   // UNICODE_TO_GBK[4694] := 16#545E;
   // UNICODE_TO_GBK[4695] := 16#85DA;
   // UNICODE_TO_GBK[4696] := 16#545F;
   // UNICODE_TO_GBK[4697] := 16#85DB;
   // UNICODE_TO_GBK[4698] := 16#5460;
   // UNICODE_TO_GBK[4699] := 16#85DC;
   // UNICODE_TO_GBK[4700] := 16#5461;
   // UNICODE_TO_GBK[4701] := 16#85DD;
   // UNICODE_TO_GBK[4702] := 16#5462;
   // UNICODE_TO_GBK[4703] := 16#C4D8;
   // UNICODE_TO_GBK[4704] := 16#5463;
   // UNICODE_TO_GBK[4705] := 16#85DE;
   // UNICODE_TO_GBK[4706] := 16#5464;
   // UNICODE_TO_GBK[4707] := 16#DFCA;
   // UNICODE_TO_GBK[4708] := 16#5465;
   // UNICODE_TO_GBK[4709] := 16#85DF;
   // UNICODE_TO_GBK[4710] := 16#5466;
   // UNICODE_TO_GBK[4711] := 16#DFCF;
   // UNICODE_TO_GBK[4712] := 16#5467;
   // UNICODE_TO_GBK[4713] := 16#85E0;
   // UNICODE_TO_GBK[4714] := 16#5468;
   // UNICODE_TO_GBK[4715] := 16#D6DC;
   // UNICODE_TO_GBK[4716] := 16#5469;
   // UNICODE_TO_GBK[4717] := 16#85E1;
   // UNICODE_TO_GBK[4718] := 16#546A;
   // UNICODE_TO_GBK[4719] := 16#85E2;
   // UNICODE_TO_GBK[4720] := 16#546B;
   // UNICODE_TO_GBK[4721] := 16#85E3;
   // UNICODE_TO_GBK[4722] := 16#546C;
   // UNICODE_TO_GBK[4723] := 16#85E4;
   // UNICODE_TO_GBK[4724] := 16#546D;
   // UNICODE_TO_GBK[4725] := 16#85E5;
   // UNICODE_TO_GBK[4726] := 16#546E;
   // UNICODE_TO_GBK[4727] := 16#85E6;
   // UNICODE_TO_GBK[4728] := 16#546F;
   // UNICODE_TO_GBK[4729] := 16#85E7;
   // UNICODE_TO_GBK[4730] := 16#5470;
   // UNICODE_TO_GBK[4731] := 16#85E8;
   // UNICODE_TO_GBK[4732] := 16#5471;
   // UNICODE_TO_GBK[4733] := 16#DFC9;
   // UNICODE_TO_GBK[4734] := 16#5472;
   // UNICODE_TO_GBK[4735] := 16#DFDA;
   // UNICODE_TO_GBK[4736] := 16#5473;
   // UNICODE_TO_GBK[4737] := 16#CEB6;
   // UNICODE_TO_GBK[4738] := 16#5474;
   // UNICODE_TO_GBK[4739] := 16#85E9;
   // UNICODE_TO_GBK[4740] := 16#5475;
   // UNICODE_TO_GBK[4741] := 16#BAC7;
   // UNICODE_TO_GBK[4742] := 16#5476;
   // UNICODE_TO_GBK[4743] := 16#DFCE;
   // UNICODE_TO_GBK[4744] := 16#5477;
   // UNICODE_TO_GBK[4745] := 16#DFC8;
   // UNICODE_TO_GBK[4746] := 16#5478;
   // UNICODE_TO_GBK[4747] := 16#C5DE;
   // UNICODE_TO_GBK[4748] := 16#5479;
   // UNICODE_TO_GBK[4749] := 16#85EA;
   // UNICODE_TO_GBK[4750] := 16#547A;
   // UNICODE_TO_GBK[4751] := 16#85EB;
   // UNICODE_TO_GBK[4752] := 16#547B;
   // UNICODE_TO_GBK[4753] := 16#C9EB;
   // UNICODE_TO_GBK[4754] := 16#547C;
   // UNICODE_TO_GBK[4755] := 16#BAF4;
   // UNICODE_TO_GBK[4756] := 16#547D;
   // UNICODE_TO_GBK[4757] := 16#C3FC;
   // UNICODE_TO_GBK[4758] := 16#547E;
   // UNICODE_TO_GBK[4759] := 16#85EC;
   // UNICODE_TO_GBK[4760] := 16#547F;
   // UNICODE_TO_GBK[4761] := 16#85ED;
   // UNICODE_TO_GBK[4762] := 16#5480;
   // UNICODE_TO_GBK[4763] := 16#BED7;
   // UNICODE_TO_GBK[4764] := 16#5481;
   // UNICODE_TO_GBK[4765] := 16#85EE;
   // UNICODE_TO_GBK[4766] := 16#5482;
   // UNICODE_TO_GBK[4767] := 16#DFC6;
   // UNICODE_TO_GBK[4768] := 16#5483;
   // UNICODE_TO_GBK[4769] := 16#85EF;
   // UNICODE_TO_GBK[4770] := 16#5484;
   // UNICODE_TO_GBK[4771] := 16#DFCD;
   // UNICODE_TO_GBK[4772] := 16#5485;
   // UNICODE_TO_GBK[4773] := 16#85F0;
   // UNICODE_TO_GBK[4774] := 16#5486;
   // UNICODE_TO_GBK[4775] := 16#C5D8;
   // UNICODE_TO_GBK[4776] := 16#5487;
   // UNICODE_TO_GBK[4777] := 16#85F1;
   // UNICODE_TO_GBK[4778] := 16#5488;
   // UNICODE_TO_GBK[4779] := 16#85F2;
   // UNICODE_TO_GBK[4780] := 16#5489;
   // UNICODE_TO_GBK[4781] := 16#85F3;
   // UNICODE_TO_GBK[4782] := 16#548A;
   // UNICODE_TO_GBK[4783] := 16#85F4;
   // UNICODE_TO_GBK[4784] := 16#548B;
   // UNICODE_TO_GBK[4785] := 16#D5A6;
   // UNICODE_TO_GBK[4786] := 16#548C;
   // UNICODE_TO_GBK[4787] := 16#BACD;
   // UNICODE_TO_GBK[4788] := 16#548D;
   // UNICODE_TO_GBK[4789] := 16#85F5;
   // UNICODE_TO_GBK[4790] := 16#548E;
   // UNICODE_TO_GBK[4791] := 16#BECC;
   // UNICODE_TO_GBK[4792] := 16#548F;
   // UNICODE_TO_GBK[4793] := 16#D3BD;
   // UNICODE_TO_GBK[4794] := 16#5490;
   // UNICODE_TO_GBK[4795] := 16#B8C0;
   // UNICODE_TO_GBK[4796] := 16#5491;
   // UNICODE_TO_GBK[4797] := 16#85F6;
   // UNICODE_TO_GBK[4798] := 16#5492;
   // UNICODE_TO_GBK[4799] := 16#D6E4;
   // UNICODE_TO_GBK[4800] := 16#5493;
   // UNICODE_TO_GBK[4801] := 16#85F7;
   // UNICODE_TO_GBK[4802] := 16#5494;
   // UNICODE_TO_GBK[4803] := 16#DFC7;
   // UNICODE_TO_GBK[4804] := 16#5495;
   // UNICODE_TO_GBK[4805] := 16#B9BE;
   // UNICODE_TO_GBK[4806] := 16#5496;
   // UNICODE_TO_GBK[4807] := 16#BFA7;
   // UNICODE_TO_GBK[4808] := 16#5497;
   // UNICODE_TO_GBK[4809] := 16#85F8;
   // UNICODE_TO_GBK[4810] := 16#5498;
   // UNICODE_TO_GBK[4811] := 16#85F9;
   // UNICODE_TO_GBK[4812] := 16#5499;
   // UNICODE_TO_GBK[4813] := 16#C1FC;
   // UNICODE_TO_GBK[4814] := 16#549A;
   // UNICODE_TO_GBK[4815] := 16#DFCB;
   // UNICODE_TO_GBK[4816] := 16#549B;
   // UNICODE_TO_GBK[4817] := 16#DFCC;
   // UNICODE_TO_GBK[4818] := 16#549C;
   // UNICODE_TO_GBK[4819] := 16#85FA;
   // UNICODE_TO_GBK[4820] := 16#549D;
   // UNICODE_TO_GBK[4821] := 16#DFD0;
   // UNICODE_TO_GBK[4822] := 16#549E;
   // UNICODE_TO_GBK[4823] := 16#85FB;
   // UNICODE_TO_GBK[4824] := 16#549F;
   // UNICODE_TO_GBK[4825] := 16#85FC;
   // UNICODE_TO_GBK[4826] := 16#54A0;
   // UNICODE_TO_GBK[4827] := 16#85FD;
   // UNICODE_TO_GBK[4828] := 16#54A1;
   // UNICODE_TO_GBK[4829] := 16#85FE;
   // UNICODE_TO_GBK[4830] := 16#54A2;
   // UNICODE_TO_GBK[4831] := 16#8640;
   // UNICODE_TO_GBK[4832] := 16#54A3;
   // UNICODE_TO_GBK[4833] := 16#DFDB;
   // UNICODE_TO_GBK[4834] := 16#54A4;
   // UNICODE_TO_GBK[4835] := 16#DFE5;
   // UNICODE_TO_GBK[4836] := 16#54A5;
   // UNICODE_TO_GBK[4837] := 16#8641;
   // UNICODE_TO_GBK[4838] := 16#54A6;
   // UNICODE_TO_GBK[4839] := 16#DFD7;
   // UNICODE_TO_GBK[4840] := 16#54A7;
   // UNICODE_TO_GBK[4841] := 16#DFD6;
   // UNICODE_TO_GBK[4842] := 16#54A8;
   // UNICODE_TO_GBK[4843] := 16#D7C9;
   // UNICODE_TO_GBK[4844] := 16#54A9;
   // UNICODE_TO_GBK[4845] := 16#DFE3;
   // UNICODE_TO_GBK[4846] := 16#54AA;
   // UNICODE_TO_GBK[4847] := 16#DFE4;
   // UNICODE_TO_GBK[4848] := 16#54AB;
   // UNICODE_TO_GBK[4849] := 16#E5EB;
   // UNICODE_TO_GBK[4850] := 16#54AC;
   // UNICODE_TO_GBK[4851] := 16#D2A7;
   // UNICODE_TO_GBK[4852] := 16#54AD;
   // UNICODE_TO_GBK[4853] := 16#DFD2;
   // UNICODE_TO_GBK[4854] := 16#54AE;
   // UNICODE_TO_GBK[4855] := 16#8642;
   // UNICODE_TO_GBK[4856] := 16#54AF;
   // UNICODE_TO_GBK[4857] := 16#BFA9;
   // UNICODE_TO_GBK[4858] := 16#54B0;
   // UNICODE_TO_GBK[4859] := 16#8643;
   // UNICODE_TO_GBK[4860] := 16#54B1;
   // UNICODE_TO_GBK[4861] := 16#D4DB;
   // UNICODE_TO_GBK[4862] := 16#54B2;
   // UNICODE_TO_GBK[4863] := 16#8644;
   // UNICODE_TO_GBK[4864] := 16#54B3;
   // UNICODE_TO_GBK[4865] := 16#BFC8;
   // UNICODE_TO_GBK[4866] := 16#54B4;
   // UNICODE_TO_GBK[4867] := 16#DFD4;
   // UNICODE_TO_GBK[4868] := 16#54B5;
   // UNICODE_TO_GBK[4869] := 16#8645;
   // UNICODE_TO_GBK[4870] := 16#54B6;
   // UNICODE_TO_GBK[4871] := 16#8646;
   // UNICODE_TO_GBK[4872] := 16#54B7;
   // UNICODE_TO_GBK[4873] := 16#8647;
   // UNICODE_TO_GBK[4874] := 16#54B8;
   // UNICODE_TO_GBK[4875] := 16#CFCC;
   // UNICODE_TO_GBK[4876] := 16#54B9;
   // UNICODE_TO_GBK[4877] := 16#8648;
   // UNICODE_TO_GBK[4878] := 16#54BA;
   // UNICODE_TO_GBK[4879] := 16#8649;
   // UNICODE_TO_GBK[4880] := 16#54BB;
   // UNICODE_TO_GBK[4881] := 16#DFDD;
   // UNICODE_TO_GBK[4882] := 16#54BC;
   // UNICODE_TO_GBK[4883] := 16#864A;
   // UNICODE_TO_GBK[4884] := 16#54BD;
   // UNICODE_TO_GBK[4885] := 16#D1CA;
   // UNICODE_TO_GBK[4886] := 16#54BE;
   // UNICODE_TO_GBK[4887] := 16#864B;
   // UNICODE_TO_GBK[4888] := 16#54BF;
   // UNICODE_TO_GBK[4889] := 16#DFDE;
   // UNICODE_TO_GBK[4890] := 16#54C0;
   // UNICODE_TO_GBK[4891] := 16#B0A7;
   // UNICODE_TO_GBK[4892] := 16#54C1;
   // UNICODE_TO_GBK[4893] := 16#C6B7;
   // UNICODE_TO_GBK[4894] := 16#54C2;
   // UNICODE_TO_GBK[4895] := 16#DFD3;
   // UNICODE_TO_GBK[4896] := 16#54C3;
   // UNICODE_TO_GBK[4897] := 16#864C;
   // UNICODE_TO_GBK[4898] := 16#54C4;
   // UNICODE_TO_GBK[4899] := 16#BAE5;
   // UNICODE_TO_GBK[4900] := 16#54C5;
   // UNICODE_TO_GBK[4901] := 16#864D;
   // UNICODE_TO_GBK[4902] := 16#54C6;
   // UNICODE_TO_GBK[4903] := 16#B6DF;
   // UNICODE_TO_GBK[4904] := 16#54C7;
   // UNICODE_TO_GBK[4905] := 16#CDDB;
   // UNICODE_TO_GBK[4906] := 16#54C8;
   // UNICODE_TO_GBK[4907] := 16#B9FE;
   // UNICODE_TO_GBK[4908] := 16#54C9;
   // UNICODE_TO_GBK[4909] := 16#D4D5;
   // UNICODE_TO_GBK[4910] := 16#54CA;
   // UNICODE_TO_GBK[4911] := 16#864E;
   // UNICODE_TO_GBK[4912] := 16#54CB;
   // UNICODE_TO_GBK[4913] := 16#864F;
   // UNICODE_TO_GBK[4914] := 16#54CC;
   // UNICODE_TO_GBK[4915] := 16#DFDF;
   // UNICODE_TO_GBK[4916] := 16#54CD;
   // UNICODE_TO_GBK[4917] := 16#CFEC;
   // UNICODE_TO_GBK[4918] := 16#54CE;
   // UNICODE_TO_GBK[4919] := 16#B0A5;
   // UNICODE_TO_GBK[4920] := 16#54CF;
   // UNICODE_TO_GBK[4921] := 16#DFE7;
   // UNICODE_TO_GBK[4922] := 16#54D0;
   // UNICODE_TO_GBK[4923] := 16#DFD1;
   // UNICODE_TO_GBK[4924] := 16#54D1;
   // UNICODE_TO_GBK[4925] := 16#D1C6;
   // UNICODE_TO_GBK[4926] := 16#54D2;
   // UNICODE_TO_GBK[4927] := 16#DFD5;
   // UNICODE_TO_GBK[4928] := 16#54D3;
   // UNICODE_TO_GBK[4929] := 16#DFD8;
   // UNICODE_TO_GBK[4930] := 16#54D4;
   // UNICODE_TO_GBK[4931] := 16#DFD9;
   // UNICODE_TO_GBK[4932] := 16#54D5;
   // UNICODE_TO_GBK[4933] := 16#DFDC;
   // UNICODE_TO_GBK[4934] := 16#54D6;
   // UNICODE_TO_GBK[4935] := 16#8650;
   // UNICODE_TO_GBK[4936] := 16#54D7;
   // UNICODE_TO_GBK[4937] := 16#BBA9;
   // UNICODE_TO_GBK[4938] := 16#54D8;
   // UNICODE_TO_GBK[4939] := 16#8651;
   // UNICODE_TO_GBK[4940] := 16#54D9;
   // UNICODE_TO_GBK[4941] := 16#DFE0;
   // UNICODE_TO_GBK[4942] := 16#54DA;
   // UNICODE_TO_GBK[4943] := 16#DFE1;
   // UNICODE_TO_GBK[4944] := 16#54DB;
   // UNICODE_TO_GBK[4945] := 16#8652;
   // UNICODE_TO_GBK[4946] := 16#54DC;
   // UNICODE_TO_GBK[4947] := 16#DFE2;
   // UNICODE_TO_GBK[4948] := 16#54DD;
   // UNICODE_TO_GBK[4949] := 16#DFE6;
   // UNICODE_TO_GBK[4950] := 16#54DE;
   // UNICODE_TO_GBK[4951] := 16#DFE8;
   // UNICODE_TO_GBK[4952] := 16#54DF;
   // UNICODE_TO_GBK[4953] := 16#D3B4;
   // UNICODE_TO_GBK[4954] := 16#54E0;
   // UNICODE_TO_GBK[4955] := 16#8653;
   // UNICODE_TO_GBK[4956] := 16#54E1;
   // UNICODE_TO_GBK[4957] := 16#8654;
   // UNICODE_TO_GBK[4958] := 16#54E2;
   // UNICODE_TO_GBK[4959] := 16#8655;
   // UNICODE_TO_GBK[4960] := 16#54E3;
   // UNICODE_TO_GBK[4961] := 16#8656;
   // UNICODE_TO_GBK[4962] := 16#54E4;
   // UNICODE_TO_GBK[4963] := 16#8657;
   // UNICODE_TO_GBK[4964] := 16#54E5;
   // UNICODE_TO_GBK[4965] := 16#B8E7;
   // UNICODE_TO_GBK[4966] := 16#54E6;
   // UNICODE_TO_GBK[4967] := 16#C5B6;
   // UNICODE_TO_GBK[4968] := 16#54E7;
   // UNICODE_TO_GBK[4969] := 16#DFEA;
   // UNICODE_TO_GBK[4970] := 16#54E8;
   // UNICODE_TO_GBK[4971] := 16#C9DA;
   // UNICODE_TO_GBK[4972] := 16#54E9;
   // UNICODE_TO_GBK[4973] := 16#C1A8;
   // UNICODE_TO_GBK[4974] := 16#54EA;
   // UNICODE_TO_GBK[4975] := 16#C4C4;
   // UNICODE_TO_GBK[4976] := 16#54EB;
   // UNICODE_TO_GBK[4977] := 16#8658;
   // UNICODE_TO_GBK[4978] := 16#54EC;
   // UNICODE_TO_GBK[4979] := 16#8659;
   // UNICODE_TO_GBK[4980] := 16#54ED;
   // UNICODE_TO_GBK[4981] := 16#BFDE;
   // UNICODE_TO_GBK[4982] := 16#54EE;
   // UNICODE_TO_GBK[4983] := 16#CFF8;
   // UNICODE_TO_GBK[4984] := 16#54EF;
   // UNICODE_TO_GBK[4985] := 16#865A;
   // UNICODE_TO_GBK[4986] := 16#54F0;
   // UNICODE_TO_GBK[4987] := 16#865B;
   // UNICODE_TO_GBK[4988] := 16#54F1;
   // UNICODE_TO_GBK[4989] := 16#865C;
   // UNICODE_TO_GBK[4990] := 16#54F2;
   // UNICODE_TO_GBK[4991] := 16#D5DC;
   // UNICODE_TO_GBK[4992] := 16#54F3;
   // UNICODE_TO_GBK[4993] := 16#DFEE;
   // UNICODE_TO_GBK[4994] := 16#54F4;
   // UNICODE_TO_GBK[4995] := 16#865D;
   // UNICODE_TO_GBK[4996] := 16#54F5;
   // UNICODE_TO_GBK[4997] := 16#865E;
   // UNICODE_TO_GBK[4998] := 16#54F6;
   // UNICODE_TO_GBK[4999] := 16#865F;
   // UNICODE_TO_GBK[5000] := 16#54F7;
   // UNICODE_TO_GBK[5001] := 16#8660;
   // UNICODE_TO_GBK[5002] := 16#54F8;
   // UNICODE_TO_GBK[5003] := 16#8661;
   // UNICODE_TO_GBK[5004] := 16#54F9;
   // UNICODE_TO_GBK[5005] := 16#8662;
   // UNICODE_TO_GBK[5006] := 16#54FA;
   // UNICODE_TO_GBK[5007] := 16#B2B8;
   // UNICODE_TO_GBK[5008] := 16#54FB;
   // UNICODE_TO_GBK[5009] := 16#8663;
   // UNICODE_TO_GBK[5010] := 16#54FC;
   // UNICODE_TO_GBK[5011] := 16#BADF;
   // UNICODE_TO_GBK[5012] := 16#54FD;
   // UNICODE_TO_GBK[5013] := 16#DFEC;
   // UNICODE_TO_GBK[5014] := 16#54FE;
   // UNICODE_TO_GBK[5015] := 16#8664;
   // UNICODE_TO_GBK[5016] := 16#54FF;
   // UNICODE_TO_GBK[5017] := 16#DBC1;
   // UNICODE_TO_GBK[5018] := 16#5500;
   // UNICODE_TO_GBK[5019] := 16#8665;
   // UNICODE_TO_GBK[5020] := 16#5501;
   // UNICODE_TO_GBK[5021] := 16#D1E4;
   // UNICODE_TO_GBK[5022] := 16#5502;
   // UNICODE_TO_GBK[5023] := 16#8666;
   // UNICODE_TO_GBK[5024] := 16#5503;
   // UNICODE_TO_GBK[5025] := 16#8667;
   // UNICODE_TO_GBK[5026] := 16#5504;
   // UNICODE_TO_GBK[5027] := 16#8668;
   // UNICODE_TO_GBK[5028] := 16#5505;
   // UNICODE_TO_GBK[5029] := 16#8669;
   // UNICODE_TO_GBK[5030] := 16#5506;
   // UNICODE_TO_GBK[5031] := 16#CBF4;
   // UNICODE_TO_GBK[5032] := 16#5507;
   // UNICODE_TO_GBK[5033] := 16#B4BD;
   // UNICODE_TO_GBK[5034] := 16#5508;
   // UNICODE_TO_GBK[5035] := 16#866A;
   // UNICODE_TO_GBK[5036] := 16#5509;
   // UNICODE_TO_GBK[5037] := 16#B0A6;
   // UNICODE_TO_GBK[5038] := 16#550A;
   // UNICODE_TO_GBK[5039] := 16#866B;
   // UNICODE_TO_GBK[5040] := 16#550B;
   // UNICODE_TO_GBK[5041] := 16#866C;
   // UNICODE_TO_GBK[5042] := 16#550C;
   // UNICODE_TO_GBK[5043] := 16#866D;
   // UNICODE_TO_GBK[5044] := 16#550D;
   // UNICODE_TO_GBK[5045] := 16#866E;
   // UNICODE_TO_GBK[5046] := 16#550E;
   // UNICODE_TO_GBK[5047] := 16#866F;
   // UNICODE_TO_GBK[5048] := 16#550F;
   // UNICODE_TO_GBK[5049] := 16#DFF1;
   // UNICODE_TO_GBK[5050] := 16#5510;
   // UNICODE_TO_GBK[5051] := 16#CCC6;
   // UNICODE_TO_GBK[5052] := 16#5511;
   // UNICODE_TO_GBK[5053] := 16#DFF2;
   // UNICODE_TO_GBK[5054] := 16#5512;
   // UNICODE_TO_GBK[5055] := 16#8670;
   // UNICODE_TO_GBK[5056] := 16#5513;
   // UNICODE_TO_GBK[5057] := 16#8671;
   // UNICODE_TO_GBK[5058] := 16#5514;
   // UNICODE_TO_GBK[5059] := 16#DFED;
   // UNICODE_TO_GBK[5060] := 16#5515;
   // UNICODE_TO_GBK[5061] := 16#8672;
   // UNICODE_TO_GBK[5062] := 16#5516;
   // UNICODE_TO_GBK[5063] := 16#8673;
   // UNICODE_TO_GBK[5064] := 16#5517;
   // UNICODE_TO_GBK[5065] := 16#8674;
   // UNICODE_TO_GBK[5066] := 16#5518;
   // UNICODE_TO_GBK[5067] := 16#8675;
   // UNICODE_TO_GBK[5068] := 16#5519;
   // UNICODE_TO_GBK[5069] := 16#8676;
   // UNICODE_TO_GBK[5070] := 16#551A;
   // UNICODE_TO_GBK[5071] := 16#8677;
   // UNICODE_TO_GBK[5072] := 16#551B;
   // UNICODE_TO_GBK[5073] := 16#DFE9;
   // UNICODE_TO_GBK[5074] := 16#551C;
   // UNICODE_TO_GBK[5075] := 16#8678;
   // UNICODE_TO_GBK[5076] := 16#551D;
   // UNICODE_TO_GBK[5077] := 16#8679;
   // UNICODE_TO_GBK[5078] := 16#551E;
   // UNICODE_TO_GBK[5079] := 16#867A;
   // UNICODE_TO_GBK[5080] := 16#551F;
   // UNICODE_TO_GBK[5081] := 16#867B;
   // UNICODE_TO_GBK[5082] := 16#5520;
   // UNICODE_TO_GBK[5083] := 16#DFEB;
   // UNICODE_TO_GBK[5084] := 16#5521;
   // UNICODE_TO_GBK[5085] := 16#867C;
   // UNICODE_TO_GBK[5086] := 16#5522;
   // UNICODE_TO_GBK[5087] := 16#DFEF;
   // UNICODE_TO_GBK[5088] := 16#5523;
   // UNICODE_TO_GBK[5089] := 16#DFF0;
   // UNICODE_TO_GBK[5090] := 16#5524;
   // UNICODE_TO_GBK[5091] := 16#BBBD;
   // UNICODE_TO_GBK[5092] := 16#5525;
   // UNICODE_TO_GBK[5093] := 16#867D;
   // UNICODE_TO_GBK[5094] := 16#5526;
   // UNICODE_TO_GBK[5095] := 16#867E;
   // UNICODE_TO_GBK[5096] := 16#5527;
   // UNICODE_TO_GBK[5097] := 16#DFF3;
   // UNICODE_TO_GBK[5098] := 16#5528;
   // UNICODE_TO_GBK[5099] := 16#8680;
   // UNICODE_TO_GBK[5100] := 16#5529;
   // UNICODE_TO_GBK[5101] := 16#8681;
   // UNICODE_TO_GBK[5102] := 16#552A;
   // UNICODE_TO_GBK[5103] := 16#DFF4;
   // UNICODE_TO_GBK[5104] := 16#552B;
   // UNICODE_TO_GBK[5105] := 16#8682;
   // UNICODE_TO_GBK[5106] := 16#552C;
   // UNICODE_TO_GBK[5107] := 16#BBA3;
   // UNICODE_TO_GBK[5108] := 16#552D;
   // UNICODE_TO_GBK[5109] := 16#8683;
   // UNICODE_TO_GBK[5110] := 16#552E;
   // UNICODE_TO_GBK[5111] := 16#CADB;
   // UNICODE_TO_GBK[5112] := 16#552F;
   // UNICODE_TO_GBK[5113] := 16#CEA8;
   // UNICODE_TO_GBK[5114] := 16#5530;
   // UNICODE_TO_GBK[5115] := 16#E0A7;
   // UNICODE_TO_GBK[5116] := 16#5531;
   // UNICODE_TO_GBK[5117] := 16#B3AA;
   // UNICODE_TO_GBK[5118] := 16#5532;
   // UNICODE_TO_GBK[5119] := 16#8684;
   // UNICODE_TO_GBK[5120] := 16#5533;
   // UNICODE_TO_GBK[5121] := 16#E0A6;
   // UNICODE_TO_GBK[5122] := 16#5534;
   // UNICODE_TO_GBK[5123] := 16#8685;
   // UNICODE_TO_GBK[5124] := 16#5535;
   // UNICODE_TO_GBK[5125] := 16#8686;
   // UNICODE_TO_GBK[5126] := 16#5536;
   // UNICODE_TO_GBK[5127] := 16#8687;
   // UNICODE_TO_GBK[5128] := 16#5537;
   // UNICODE_TO_GBK[5129] := 16#E0A1;
   // UNICODE_TO_GBK[5130] := 16#5538;
   // UNICODE_TO_GBK[5131] := 16#8688;
   // UNICODE_TO_GBK[5132] := 16#5539;
   // UNICODE_TO_GBK[5133] := 16#8689;
   // UNICODE_TO_GBK[5134] := 16#553A;
   // UNICODE_TO_GBK[5135] := 16#868A;
   // UNICODE_TO_GBK[5136] := 16#553B;
   // UNICODE_TO_GBK[5137] := 16#868B;
   // UNICODE_TO_GBK[5138] := 16#553C;
   // UNICODE_TO_GBK[5139] := 16#DFFE;
   // UNICODE_TO_GBK[5140] := 16#553D;
   // UNICODE_TO_GBK[5141] := 16#868C;
   // UNICODE_TO_GBK[5142] := 16#553E;
   // UNICODE_TO_GBK[5143] := 16#CDD9;
   // UNICODE_TO_GBK[5144] := 16#553F;
   // UNICODE_TO_GBK[5145] := 16#DFFC;
   // UNICODE_TO_GBK[5146] := 16#5540;
   // UNICODE_TO_GBK[5147] := 16#868D;
   // UNICODE_TO_GBK[5148] := 16#5541;
   // UNICODE_TO_GBK[5149] := 16#DFFA;
   // UNICODE_TO_GBK[5150] := 16#5542;
   // UNICODE_TO_GBK[5151] := 16#868E;
   // UNICODE_TO_GBK[5152] := 16#5543;
   // UNICODE_TO_GBK[5153] := 16#BFD0;
   // UNICODE_TO_GBK[5154] := 16#5544;
   // UNICODE_TO_GBK[5155] := 16#D7C4;
   // UNICODE_TO_GBK[5156] := 16#5545;
   // UNICODE_TO_GBK[5157] := 16#868F;
   // UNICODE_TO_GBK[5158] := 16#5546;
   // UNICODE_TO_GBK[5159] := 16#C9CC;
   // UNICODE_TO_GBK[5160] := 16#5547;
   // UNICODE_TO_GBK[5161] := 16#8690;
   // UNICODE_TO_GBK[5162] := 16#5548;
   // UNICODE_TO_GBK[5163] := 16#8691;
   // UNICODE_TO_GBK[5164] := 16#5549;
   // UNICODE_TO_GBK[5165] := 16#DFF8;
   // UNICODE_TO_GBK[5166] := 16#554A;
   // UNICODE_TO_GBK[5167] := 16#B0A1;
   // UNICODE_TO_GBK[5168] := 16#554B;
   // UNICODE_TO_GBK[5169] := 16#8692;
   // UNICODE_TO_GBK[5170] := 16#554C;
   // UNICODE_TO_GBK[5171] := 16#8693;
   // UNICODE_TO_GBK[5172] := 16#554D;
   // UNICODE_TO_GBK[5173] := 16#8694;
   // UNICODE_TO_GBK[5174] := 16#554E;
   // UNICODE_TO_GBK[5175] := 16#8695;
   // UNICODE_TO_GBK[5176] := 16#554F;
   // UNICODE_TO_GBK[5177] := 16#8696;
   // UNICODE_TO_GBK[5178] := 16#5550;
   // UNICODE_TO_GBK[5179] := 16#DFFD;
   // UNICODE_TO_GBK[5180] := 16#5551;
   // UNICODE_TO_GBK[5181] := 16#8697;
   // UNICODE_TO_GBK[5182] := 16#5552;
   // UNICODE_TO_GBK[5183] := 16#8698;
   // UNICODE_TO_GBK[5184] := 16#5553;
   // UNICODE_TO_GBK[5185] := 16#8699;
   // UNICODE_TO_GBK[5186] := 16#5554;
   // UNICODE_TO_GBK[5187] := 16#869A;
   // UNICODE_TO_GBK[5188] := 16#5555;
   // UNICODE_TO_GBK[5189] := 16#DFFB;
   // UNICODE_TO_GBK[5190] := 16#5556;
   // UNICODE_TO_GBK[5191] := 16#E0A2;
   // UNICODE_TO_GBK[5192] := 16#5557;
   // UNICODE_TO_GBK[5193] := 16#869B;
   // UNICODE_TO_GBK[5194] := 16#5558;
   // UNICODE_TO_GBK[5195] := 16#869C;
   // UNICODE_TO_GBK[5196] := 16#5559;
   // UNICODE_TO_GBK[5197] := 16#869D;
   // UNICODE_TO_GBK[5198] := 16#555A;
   // UNICODE_TO_GBK[5199] := 16#869E;
   // UNICODE_TO_GBK[5200] := 16#555B;
   // UNICODE_TO_GBK[5201] := 16#869F;
   // UNICODE_TO_GBK[5202] := 16#555C;
   // UNICODE_TO_GBK[5203] := 16#E0A8;
   // UNICODE_TO_GBK[5204] := 16#555D;
   // UNICODE_TO_GBK[5205] := 16#86A0;
   // UNICODE_TO_GBK[5206] := 16#555E;
   // UNICODE_TO_GBK[5207] := 16#86A1;
   // UNICODE_TO_GBK[5208] := 16#555F;
   // UNICODE_TO_GBK[5209] := 16#86A2;
   // UNICODE_TO_GBK[5210] := 16#5560;
   // UNICODE_TO_GBK[5211] := 16#86A3;
   // UNICODE_TO_GBK[5212] := 16#5561;
   // UNICODE_TO_GBK[5213] := 16#B7C8;
   // UNICODE_TO_GBK[5214] := 16#5562;
   // UNICODE_TO_GBK[5215] := 16#86A4;
   // UNICODE_TO_GBK[5216] := 16#5563;
   // UNICODE_TO_GBK[5217] := 16#86A5;
   // UNICODE_TO_GBK[5218] := 16#5564;
   // UNICODE_TO_GBK[5219] := 16#C6A1;
   // UNICODE_TO_GBK[5220] := 16#5565;
   // UNICODE_TO_GBK[5221] := 16#C9B6;
   // UNICODE_TO_GBK[5222] := 16#5566;
   // UNICODE_TO_GBK[5223] := 16#C0B2;
   // UNICODE_TO_GBK[5224] := 16#5567;
   // UNICODE_TO_GBK[5225] := 16#DFF5;
   // UNICODE_TO_GBK[5226] := 16#5568;
   // UNICODE_TO_GBK[5227] := 16#86A6;
   // UNICODE_TO_GBK[5228] := 16#5569;
   // UNICODE_TO_GBK[5229] := 16#86A7;
   // UNICODE_TO_GBK[5230] := 16#556A;
   // UNICODE_TO_GBK[5231] := 16#C5BE;
   // UNICODE_TO_GBK[5232] := 16#556B;
   // UNICODE_TO_GBK[5233] := 16#86A8;
   // UNICODE_TO_GBK[5234] := 16#556C;
   // UNICODE_TO_GBK[5235] := 16#D8C4;
   // UNICODE_TO_GBK[5236] := 16#556D;
   // UNICODE_TO_GBK[5237] := 16#DFF9;
   // UNICODE_TO_GBK[5238] := 16#556E;
   // UNICODE_TO_GBK[5239] := 16#C4F6;
   // UNICODE_TO_GBK[5240] := 16#556F;
   // UNICODE_TO_GBK[5241] := 16#86A9;
   // UNICODE_TO_GBK[5242] := 16#5570;
   // UNICODE_TO_GBK[5243] := 16#86AA;
   // UNICODE_TO_GBK[5244] := 16#5571;
   // UNICODE_TO_GBK[5245] := 16#86AB;
   // UNICODE_TO_GBK[5246] := 16#5572;
   // UNICODE_TO_GBK[5247] := 16#86AC;
   // UNICODE_TO_GBK[5248] := 16#5573;
   // UNICODE_TO_GBK[5249] := 16#86AD;
   // UNICODE_TO_GBK[5250] := 16#5574;
   // UNICODE_TO_GBK[5251] := 16#86AE;
   // UNICODE_TO_GBK[5252] := 16#5575;
   // UNICODE_TO_GBK[5253] := 16#E0A3;
   // UNICODE_TO_GBK[5254] := 16#5576;
   // UNICODE_TO_GBK[5255] := 16#E0A4;
   // UNICODE_TO_GBK[5256] := 16#5577;
   // UNICODE_TO_GBK[5257] := 16#E0A5;
   // UNICODE_TO_GBK[5258] := 16#5578;
   // UNICODE_TO_GBK[5259] := 16#D0A5;
   // UNICODE_TO_GBK[5260] := 16#5579;
   // UNICODE_TO_GBK[5261] := 16#86AF;
   // UNICODE_TO_GBK[5262] := 16#557A;
   // UNICODE_TO_GBK[5263] := 16#86B0;
   // UNICODE_TO_GBK[5264] := 16#557B;
   // UNICODE_TO_GBK[5265] := 16#E0B4;
   // UNICODE_TO_GBK[5266] := 16#557C;
   // UNICODE_TO_GBK[5267] := 16#CCE4;
   // UNICODE_TO_GBK[5268] := 16#557D;
   // UNICODE_TO_GBK[5269] := 16#86B1;
   // UNICODE_TO_GBK[5270] := 16#557E;
   // UNICODE_TO_GBK[5271] := 16#E0B1;
   // UNICODE_TO_GBK[5272] := 16#557F;
   // UNICODE_TO_GBK[5273] := 16#86B2;
   // UNICODE_TO_GBK[5274] := 16#5580;
   // UNICODE_TO_GBK[5275] := 16#BFA6;
   // UNICODE_TO_GBK[5276] := 16#5581;
   // UNICODE_TO_GBK[5277] := 16#E0AF;
   // UNICODE_TO_GBK[5278] := 16#5582;
   // UNICODE_TO_GBK[5279] := 16#CEB9;
   // UNICODE_TO_GBK[5280] := 16#5583;
   // UNICODE_TO_GBK[5281] := 16#E0AB;
   // UNICODE_TO_GBK[5282] := 16#5584;
   // UNICODE_TO_GBK[5283] := 16#C9C6;
   // UNICODE_TO_GBK[5284] := 16#5585;
   // UNICODE_TO_GBK[5285] := 16#86B3;
   // UNICODE_TO_GBK[5286] := 16#5586;
   // UNICODE_TO_GBK[5287] := 16#86B4;
   // UNICODE_TO_GBK[5288] := 16#5587;
   // UNICODE_TO_GBK[5289] := 16#C0AE;
   // UNICODE_TO_GBK[5290] := 16#5588;
   // UNICODE_TO_GBK[5291] := 16#E0AE;
   // UNICODE_TO_GBK[5292] := 16#5589;
   // UNICODE_TO_GBK[5293] := 16#BAED;
   // UNICODE_TO_GBK[5294] := 16#558A;
   // UNICODE_TO_GBK[5295] := 16#BAB0;
   // UNICODE_TO_GBK[5296] := 16#558B;
   // UNICODE_TO_GBK[5297] := 16#E0A9;
   // UNICODE_TO_GBK[5298] := 16#558C;
   // UNICODE_TO_GBK[5299] := 16#86B5;
   // UNICODE_TO_GBK[5300] := 16#558D;
   // UNICODE_TO_GBK[5301] := 16#86B6;
   // UNICODE_TO_GBK[5302] := 16#558E;
   // UNICODE_TO_GBK[5303] := 16#86B7;
   // UNICODE_TO_GBK[5304] := 16#558F;
   // UNICODE_TO_GBK[5305] := 16#DFF6;
   // UNICODE_TO_GBK[5306] := 16#5590;
   // UNICODE_TO_GBK[5307] := 16#86B8;
   // UNICODE_TO_GBK[5308] := 16#5591;
   // UNICODE_TO_GBK[5309] := 16#E0B3;
   // UNICODE_TO_GBK[5310] := 16#5592;
   // UNICODE_TO_GBK[5311] := 16#86B9;
   // UNICODE_TO_GBK[5312] := 16#5593;
   // UNICODE_TO_GBK[5313] := 16#86BA;
   // UNICODE_TO_GBK[5314] := 16#5594;
   // UNICODE_TO_GBK[5315] := 16#E0B8;
   // UNICODE_TO_GBK[5316] := 16#5595;
   // UNICODE_TO_GBK[5317] := 16#86BB;
   // UNICODE_TO_GBK[5318] := 16#5596;
   // UNICODE_TO_GBK[5319] := 16#86BC;
   // UNICODE_TO_GBK[5320] := 16#5597;
   // UNICODE_TO_GBK[5321] := 16#86BD;
   // UNICODE_TO_GBK[5322] := 16#5598;
   // UNICODE_TO_GBK[5323] := 16#B4AD;
   // UNICODE_TO_GBK[5324] := 16#5599;
   // UNICODE_TO_GBK[5325] := 16#E0B9;
   // UNICODE_TO_GBK[5326] := 16#559A;
   // UNICODE_TO_GBK[5327] := 16#86BE;
   // UNICODE_TO_GBK[5328] := 16#559B;
   // UNICODE_TO_GBK[5329] := 16#86BF;
   // UNICODE_TO_GBK[5330] := 16#559C;
   // UNICODE_TO_GBK[5331] := 16#CFB2;
   // UNICODE_TO_GBK[5332] := 16#559D;
   // UNICODE_TO_GBK[5333] := 16#BAC8;
   // UNICODE_TO_GBK[5334] := 16#559E;
   // UNICODE_TO_GBK[5335] := 16#86C0;
   // UNICODE_TO_GBK[5336] := 16#559F;
   // UNICODE_TO_GBK[5337] := 16#E0B0;
   // UNICODE_TO_GBK[5338] := 16#55A0;
   // UNICODE_TO_GBK[5339] := 16#86C1;
   // UNICODE_TO_GBK[5340] := 16#55A1;
   // UNICODE_TO_GBK[5341] := 16#86C2;
   // UNICODE_TO_GBK[5342] := 16#55A2;
   // UNICODE_TO_GBK[5343] := 16#86C3;
   // UNICODE_TO_GBK[5344] := 16#55A3;
   // UNICODE_TO_GBK[5345] := 16#86C4;
   // UNICODE_TO_GBK[5346] := 16#55A4;
   // UNICODE_TO_GBK[5347] := 16#86C5;
   // UNICODE_TO_GBK[5348] := 16#55A5;
   // UNICODE_TO_GBK[5349] := 16#86C6;
   // UNICODE_TO_GBK[5350] := 16#55A6;
   // UNICODE_TO_GBK[5351] := 16#86C7;
   // UNICODE_TO_GBK[5352] := 16#55A7;
   // UNICODE_TO_GBK[5353] := 16#D0FA;
   // UNICODE_TO_GBK[5354] := 16#55A8;
   // UNICODE_TO_GBK[5355] := 16#86C8;
   // UNICODE_TO_GBK[5356] := 16#55A9;
   // UNICODE_TO_GBK[5357] := 16#86C9;
   // UNICODE_TO_GBK[5358] := 16#55AA;
   // UNICODE_TO_GBK[5359] := 16#86CA;
   // UNICODE_TO_GBK[5360] := 16#55AB;
   // UNICODE_TO_GBK[5361] := 16#86CB;
   // UNICODE_TO_GBK[5362] := 16#55AC;
   // UNICODE_TO_GBK[5363] := 16#86CC;
   // UNICODE_TO_GBK[5364] := 16#55AD;
   // UNICODE_TO_GBK[5365] := 16#86CD;
   // UNICODE_TO_GBK[5366] := 16#55AE;
   // UNICODE_TO_GBK[5367] := 16#86CE;
   // UNICODE_TO_GBK[5368] := 16#55AF;
   // UNICODE_TO_GBK[5369] := 16#86CF;
   // UNICODE_TO_GBK[5370] := 16#55B0;
   // UNICODE_TO_GBK[5371] := 16#86D0;
   // UNICODE_TO_GBK[5372] := 16#55B1;
   // UNICODE_TO_GBK[5373] := 16#E0AC;
   // UNICODE_TO_GBK[5374] := 16#55B2;
   // UNICODE_TO_GBK[5375] := 16#86D1;
   // UNICODE_TO_GBK[5376] := 16#55B3;
   // UNICODE_TO_GBK[5377] := 16#D4FB;
   // UNICODE_TO_GBK[5378] := 16#55B4;
   // UNICODE_TO_GBK[5379] := 16#86D2;
   // UNICODE_TO_GBK[5380] := 16#55B5;
   // UNICODE_TO_GBK[5381] := 16#DFF7;
   // UNICODE_TO_GBK[5382] := 16#55B6;
   // UNICODE_TO_GBK[5383] := 16#86D3;
   // UNICODE_TO_GBK[5384] := 16#55B7;
   // UNICODE_TO_GBK[5385] := 16#C5E7;
   // UNICODE_TO_GBK[5386] := 16#55B8;
   // UNICODE_TO_GBK[5387] := 16#86D4;
   // UNICODE_TO_GBK[5388] := 16#55B9;
   // UNICODE_TO_GBK[5389] := 16#E0AD;
   // UNICODE_TO_GBK[5390] := 16#55BA;
   // UNICODE_TO_GBK[5391] := 16#86D5;
   // UNICODE_TO_GBK[5392] := 16#55BB;
   // UNICODE_TO_GBK[5393] := 16#D3F7;
   // UNICODE_TO_GBK[5394] := 16#55BC;
   // UNICODE_TO_GBK[5395] := 16#86D6;
   // UNICODE_TO_GBK[5396] := 16#55BD;
   // UNICODE_TO_GBK[5397] := 16#E0B6;
   // UNICODE_TO_GBK[5398] := 16#55BE;
   // UNICODE_TO_GBK[5399] := 16#E0B7;
   // UNICODE_TO_GBK[5400] := 16#55BF;
   // UNICODE_TO_GBK[5401] := 16#86D7;
   // UNICODE_TO_GBK[5402] := 16#55C0;
   // UNICODE_TO_GBK[5403] := 16#86D8;
   // UNICODE_TO_GBK[5404] := 16#55C1;
   // UNICODE_TO_GBK[5405] := 16#86D9;
   // UNICODE_TO_GBK[5406] := 16#55C2;
   // UNICODE_TO_GBK[5407] := 16#86DA;
   // UNICODE_TO_GBK[5408] := 16#55C3;
   // UNICODE_TO_GBK[5409] := 16#86DB;
   // UNICODE_TO_GBK[5410] := 16#55C4;
   // UNICODE_TO_GBK[5411] := 16#E0C4;
   // UNICODE_TO_GBK[5412] := 16#55C5;
   // UNICODE_TO_GBK[5413] := 16#D0E1;
   // UNICODE_TO_GBK[5414] := 16#55C6;
   // UNICODE_TO_GBK[5415] := 16#86DC;
   // UNICODE_TO_GBK[5416] := 16#55C7;
   // UNICODE_TO_GBK[5417] := 16#86DD;
   // UNICODE_TO_GBK[5418] := 16#55C8;
   // UNICODE_TO_GBK[5419] := 16#86DE;
   // UNICODE_TO_GBK[5420] := 16#55C9;
   // UNICODE_TO_GBK[5421] := 16#E0BC;
   // UNICODE_TO_GBK[5422] := 16#55CA;
   // UNICODE_TO_GBK[5423] := 16#86DF;
   // UNICODE_TO_GBK[5424] := 16#55CB;
   // UNICODE_TO_GBK[5425] := 16#86E0;
   // UNICODE_TO_GBK[5426] := 16#55CC;
   // UNICODE_TO_GBK[5427] := 16#E0C9;
   // UNICODE_TO_GBK[5428] := 16#55CD;
   // UNICODE_TO_GBK[5429] := 16#E0CA;
   // UNICODE_TO_GBK[5430] := 16#55CE;
   // UNICODE_TO_GBK[5431] := 16#86E1;
   // UNICODE_TO_GBK[5432] := 16#55CF;
   // UNICODE_TO_GBK[5433] := 16#86E2;
   // UNICODE_TO_GBK[5434] := 16#55D0;
   // UNICODE_TO_GBK[5435] := 16#86E3;
   // UNICODE_TO_GBK[5436] := 16#55D1;
   // UNICODE_TO_GBK[5437] := 16#E0BE;
   // UNICODE_TO_GBK[5438] := 16#55D2;
   // UNICODE_TO_GBK[5439] := 16#E0AA;
   // UNICODE_TO_GBK[5440] := 16#55D3;
   // UNICODE_TO_GBK[5441] := 16#C9A4;
   // UNICODE_TO_GBK[5442] := 16#55D4;
   // UNICODE_TO_GBK[5443] := 16#E0C1;
   // UNICODE_TO_GBK[5444] := 16#55D5;
   // UNICODE_TO_GBK[5445] := 16#86E4;
   // UNICODE_TO_GBK[5446] := 16#55D6;
   // UNICODE_TO_GBK[5447] := 16#E0B2;
   // UNICODE_TO_GBK[5448] := 16#55D7;
   // UNICODE_TO_GBK[5449] := 16#86E5;
   // UNICODE_TO_GBK[5450] := 16#55D8;
   // UNICODE_TO_GBK[5451] := 16#86E6;
   // UNICODE_TO_GBK[5452] := 16#55D9;
   // UNICODE_TO_GBK[5453] := 16#86E7;
   // UNICODE_TO_GBK[5454] := 16#55DA;
   // UNICODE_TO_GBK[5455] := 16#86E8;
   // UNICODE_TO_GBK[5456] := 16#55DB;
   // UNICODE_TO_GBK[5457] := 16#86E9;
   // UNICODE_TO_GBK[5458] := 16#55DC;
   // UNICODE_TO_GBK[5459] := 16#CAC8;
   // UNICODE_TO_GBK[5460] := 16#55DD;
   // UNICODE_TO_GBK[5461] := 16#E0C3;
   // UNICODE_TO_GBK[5462] := 16#55DE;
   // UNICODE_TO_GBK[5463] := 16#86EA;
   // UNICODE_TO_GBK[5464] := 16#55DF;
   // UNICODE_TO_GBK[5465] := 16#E0B5;
   // UNICODE_TO_GBK[5466] := 16#55E0;
   // UNICODE_TO_GBK[5467] := 16#86EB;
   // UNICODE_TO_GBK[5468] := 16#55E1;
   // UNICODE_TO_GBK[5469] := 16#CECB;
   // UNICODE_TO_GBK[5470] := 16#55E2;
   // UNICODE_TO_GBK[5471] := 16#86EC;
   // UNICODE_TO_GBK[5472] := 16#55E3;
   // UNICODE_TO_GBK[5473] := 16#CBC3;
   // UNICODE_TO_GBK[5474] := 16#55E4;
   // UNICODE_TO_GBK[5475] := 16#E0CD;
   // UNICODE_TO_GBK[5476] := 16#55E5;
   // UNICODE_TO_GBK[5477] := 16#E0C6;
   // UNICODE_TO_GBK[5478] := 16#55E6;
   // UNICODE_TO_GBK[5479] := 16#E0C2;
   // UNICODE_TO_GBK[5480] := 16#55E7;
   // UNICODE_TO_GBK[5481] := 16#86ED;
   // UNICODE_TO_GBK[5482] := 16#55E8;
   // UNICODE_TO_GBK[5483] := 16#E0CB;
   // UNICODE_TO_GBK[5484] := 16#55E9;
   // UNICODE_TO_GBK[5485] := 16#86EE;
   // UNICODE_TO_GBK[5486] := 16#55EA;
   // UNICODE_TO_GBK[5487] := 16#E0BA;
   // UNICODE_TO_GBK[5488] := 16#55EB;
   // UNICODE_TO_GBK[5489] := 16#E0BF;
   // UNICODE_TO_GBK[5490] := 16#55EC;
   // UNICODE_TO_GBK[5491] := 16#E0C0;
   // UNICODE_TO_GBK[5492] := 16#55ED;
   // UNICODE_TO_GBK[5493] := 16#86EF;
   // UNICODE_TO_GBK[5494] := 16#55EE;
   // UNICODE_TO_GBK[5495] := 16#86F0;
   // UNICODE_TO_GBK[5496] := 16#55EF;
   // UNICODE_TO_GBK[5497] := 16#E0C5;
   // UNICODE_TO_GBK[5498] := 16#55F0;
   // UNICODE_TO_GBK[5499] := 16#86F1;
   // UNICODE_TO_GBK[5500] := 16#55F1;
   // UNICODE_TO_GBK[5501] := 16#86F2;
   // UNICODE_TO_GBK[5502] := 16#55F2;
   // UNICODE_TO_GBK[5503] := 16#E0C7;
   // UNICODE_TO_GBK[5504] := 16#55F3;
   // UNICODE_TO_GBK[5505] := 16#E0C8;
   // UNICODE_TO_GBK[5506] := 16#55F4;
   // UNICODE_TO_GBK[5507] := 16#86F3;
   // UNICODE_TO_GBK[5508] := 16#55F5;
   // UNICODE_TO_GBK[5509] := 16#E0CC;
   // UNICODE_TO_GBK[5510] := 16#55F6;
   // UNICODE_TO_GBK[5511] := 16#86F4;
   // UNICODE_TO_GBK[5512] := 16#55F7;
   // UNICODE_TO_GBK[5513] := 16#E0BB;
   // UNICODE_TO_GBK[5514] := 16#55F8;
   // UNICODE_TO_GBK[5515] := 16#86F5;
   // UNICODE_TO_GBK[5516] := 16#55F9;
   // UNICODE_TO_GBK[5517] := 16#86F6;
   // UNICODE_TO_GBK[5518] := 16#55FA;
   // UNICODE_TO_GBK[5519] := 16#86F7;
   // UNICODE_TO_GBK[5520] := 16#55FB;
   // UNICODE_TO_GBK[5521] := 16#86F8;
   // UNICODE_TO_GBK[5522] := 16#55FC;
   // UNICODE_TO_GBK[5523] := 16#86F9;
   // UNICODE_TO_GBK[5524] := 16#55FD;
   // UNICODE_TO_GBK[5525] := 16#CBD4;
   // UNICODE_TO_GBK[5526] := 16#55FE;
   // UNICODE_TO_GBK[5527] := 16#E0D5;
   // UNICODE_TO_GBK[5528] := 16#55FF;
   // UNICODE_TO_GBK[5529] := 16#86FA;
   // UNICODE_TO_GBK[5530] := 16#5600;
   // UNICODE_TO_GBK[5531] := 16#E0D6;
   // UNICODE_TO_GBK[5532] := 16#5601;
   // UNICODE_TO_GBK[5533] := 16#E0D2;
   // UNICODE_TO_GBK[5534] := 16#5602;
   // UNICODE_TO_GBK[5535] := 16#86FB;
   // UNICODE_TO_GBK[5536] := 16#5603;
   // UNICODE_TO_GBK[5537] := 16#86FC;
   // UNICODE_TO_GBK[5538] := 16#5604;
   // UNICODE_TO_GBK[5539] := 16#86FD;
   // UNICODE_TO_GBK[5540] := 16#5605;
   // UNICODE_TO_GBK[5541] := 16#86FE;
   // UNICODE_TO_GBK[5542] := 16#5606;
   // UNICODE_TO_GBK[5543] := 16#8740;
   // UNICODE_TO_GBK[5544] := 16#5607;
   // UNICODE_TO_GBK[5545] := 16#8741;
   // UNICODE_TO_GBK[5546] := 16#5608;
   // UNICODE_TO_GBK[5547] := 16#E0D0;
   // UNICODE_TO_GBK[5548] := 16#5609;
   // UNICODE_TO_GBK[5549] := 16#BCCE;
   // UNICODE_TO_GBK[5550] := 16#560A;
   // UNICODE_TO_GBK[5551] := 16#8742;
   // UNICODE_TO_GBK[5552] := 16#560B;
   // UNICODE_TO_GBK[5553] := 16#8743;
   // UNICODE_TO_GBK[5554] := 16#560C;
   // UNICODE_TO_GBK[5555] := 16#E0D1;
   // UNICODE_TO_GBK[5556] := 16#560D;
   // UNICODE_TO_GBK[5557] := 16#8744;
   // UNICODE_TO_GBK[5558] := 16#560E;
   // UNICODE_TO_GBK[5559] := 16#B8C2;
   // UNICODE_TO_GBK[5560] := 16#560F;
   // UNICODE_TO_GBK[5561] := 16#D8C5;
   // UNICODE_TO_GBK[5562] := 16#5610;
   // UNICODE_TO_GBK[5563] := 16#8745;
   // UNICODE_TO_GBK[5564] := 16#5611;
   // UNICODE_TO_GBK[5565] := 16#8746;
   // UNICODE_TO_GBK[5566] := 16#5612;
   // UNICODE_TO_GBK[5567] := 16#8747;
   // UNICODE_TO_GBK[5568] := 16#5613;
   // UNICODE_TO_GBK[5569] := 16#8748;
   // UNICODE_TO_GBK[5570] := 16#5614;
   // UNICODE_TO_GBK[5571] := 16#8749;
   // UNICODE_TO_GBK[5572] := 16#5615;
   // UNICODE_TO_GBK[5573] := 16#874A;
   // UNICODE_TO_GBK[5574] := 16#5616;
   // UNICODE_TO_GBK[5575] := 16#874B;
   // UNICODE_TO_GBK[5576] := 16#5617;
   // UNICODE_TO_GBK[5577] := 16#874C;
   // UNICODE_TO_GBK[5578] := 16#5618;
   // UNICODE_TO_GBK[5579] := 16#D0EA;
   // UNICODE_TO_GBK[5580] := 16#5619;
   // UNICODE_TO_GBK[5581] := 16#874D;
   // UNICODE_TO_GBK[5582] := 16#561A;
   // UNICODE_TO_GBK[5583] := 16#874E;
   // UNICODE_TO_GBK[5584] := 16#561B;
   // UNICODE_TO_GBK[5585] := 16#C2EF;
   // UNICODE_TO_GBK[5586] := 16#561C;
   // UNICODE_TO_GBK[5587] := 16#874F;
   // UNICODE_TO_GBK[5588] := 16#561D;
   // UNICODE_TO_GBK[5589] := 16#8750;
   // UNICODE_TO_GBK[5590] := 16#561E;
   // UNICODE_TO_GBK[5591] := 16#E0CF;
   // UNICODE_TO_GBK[5592] := 16#561F;
   // UNICODE_TO_GBK[5593] := 16#E0BD;
   // UNICODE_TO_GBK[5594] := 16#5620;
   // UNICODE_TO_GBK[5595] := 16#8751;
   // UNICODE_TO_GBK[5596] := 16#5621;
   // UNICODE_TO_GBK[5597] := 16#8752;
   // UNICODE_TO_GBK[5598] := 16#5622;
   // UNICODE_TO_GBK[5599] := 16#8753;
   // UNICODE_TO_GBK[5600] := 16#5623;
   // UNICODE_TO_GBK[5601] := 16#E0D4;
   // UNICODE_TO_GBK[5602] := 16#5624;
   // UNICODE_TO_GBK[5603] := 16#E0D3;
   // UNICODE_TO_GBK[5604] := 16#5625;
   // UNICODE_TO_GBK[5605] := 16#8754;
   // UNICODE_TO_GBK[5606] := 16#5626;
   // UNICODE_TO_GBK[5607] := 16#8755;
   // UNICODE_TO_GBK[5608] := 16#5627;
   // UNICODE_TO_GBK[5609] := 16#E0D7;
   // UNICODE_TO_GBK[5610] := 16#5628;
   // UNICODE_TO_GBK[5611] := 16#8756;
   // UNICODE_TO_GBK[5612] := 16#5629;
   // UNICODE_TO_GBK[5613] := 16#8757;
   // UNICODE_TO_GBK[5614] := 16#562A;
   // UNICODE_TO_GBK[5615] := 16#8758;
   // UNICODE_TO_GBK[5616] := 16#562B;
   // UNICODE_TO_GBK[5617] := 16#8759;
   // UNICODE_TO_GBK[5618] := 16#562C;
   // UNICODE_TO_GBK[5619] := 16#E0DC;
   // UNICODE_TO_GBK[5620] := 16#562D;
   // UNICODE_TO_GBK[5621] := 16#E0D8;
   // UNICODE_TO_GBK[5622] := 16#562E;
   // UNICODE_TO_GBK[5623] := 16#875A;
   // UNICODE_TO_GBK[5624] := 16#562F;
   // UNICODE_TO_GBK[5625] := 16#875B;
   // UNICODE_TO_GBK[5626] := 16#5630;
   // UNICODE_TO_GBK[5627] := 16#875C;
   // UNICODE_TO_GBK[5628] := 16#5631;
   // UNICODE_TO_GBK[5629] := 16#D6F6;
   // UNICODE_TO_GBK[5630] := 16#5632;
   // UNICODE_TO_GBK[5631] := 16#B3B0;
   // UNICODE_TO_GBK[5632] := 16#5633;
   // UNICODE_TO_GBK[5633] := 16#875D;
   // UNICODE_TO_GBK[5634] := 16#5634;
   // UNICODE_TO_GBK[5635] := 16#D7EC;
   // UNICODE_TO_GBK[5636] := 16#5635;
   // UNICODE_TO_GBK[5637] := 16#875E;
   // UNICODE_TO_GBK[5638] := 16#5636;
   // UNICODE_TO_GBK[5639] := 16#CBBB;
   // UNICODE_TO_GBK[5640] := 16#5637;
   // UNICODE_TO_GBK[5641] := 16#875F;
   // UNICODE_TO_GBK[5642] := 16#5638;
   // UNICODE_TO_GBK[5643] := 16#8760;
   // UNICODE_TO_GBK[5644] := 16#5639;
   // UNICODE_TO_GBK[5645] := 16#E0DA;
   // UNICODE_TO_GBK[5646] := 16#563A;
   // UNICODE_TO_GBK[5647] := 16#8761;
   // UNICODE_TO_GBK[5648] := 16#563B;
   // UNICODE_TO_GBK[5649] := 16#CEFB;
   // UNICODE_TO_GBK[5650] := 16#563C;
   // UNICODE_TO_GBK[5651] := 16#8762;
   // UNICODE_TO_GBK[5652] := 16#563D;
   // UNICODE_TO_GBK[5653] := 16#8763;
   // UNICODE_TO_GBK[5654] := 16#563E;
   // UNICODE_TO_GBK[5655] := 16#8764;
   // UNICODE_TO_GBK[5656] := 16#563F;
   // UNICODE_TO_GBK[5657] := 16#BAD9;
   // UNICODE_TO_GBK[5658] := 16#5640;
   // UNICODE_TO_GBK[5659] := 16#8765;
   // UNICODE_TO_GBK[5660] := 16#5641;
   // UNICODE_TO_GBK[5661] := 16#8766;
   // UNICODE_TO_GBK[5662] := 16#5642;
   // UNICODE_TO_GBK[5663] := 16#8767;
   // UNICODE_TO_GBK[5664] := 16#5643;
   // UNICODE_TO_GBK[5665] := 16#8768;
   // UNICODE_TO_GBK[5666] := 16#5644;
   // UNICODE_TO_GBK[5667] := 16#8769;
   // UNICODE_TO_GBK[5668] := 16#5645;
   // UNICODE_TO_GBK[5669] := 16#876A;
   // UNICODE_TO_GBK[5670] := 16#5646;
   // UNICODE_TO_GBK[5671] := 16#876B;
   // UNICODE_TO_GBK[5672] := 16#5647;
   // UNICODE_TO_GBK[5673] := 16#876C;
   // UNICODE_TO_GBK[5674] := 16#5648;
   // UNICODE_TO_GBK[5675] := 16#876D;
   // UNICODE_TO_GBK[5676] := 16#5649;
   // UNICODE_TO_GBK[5677] := 16#876E;
   // UNICODE_TO_GBK[5678] := 16#564A;
   // UNICODE_TO_GBK[5679] := 16#876F;
   // UNICODE_TO_GBK[5680] := 16#564B;
   // UNICODE_TO_GBK[5681] := 16#8770;
   // UNICODE_TO_GBK[5682] := 16#564C;
   // UNICODE_TO_GBK[5683] := 16#E0E1;
   // UNICODE_TO_GBK[5684] := 16#564D;
   // UNICODE_TO_GBK[5685] := 16#E0DD;
   // UNICODE_TO_GBK[5686] := 16#564E;
   // UNICODE_TO_GBK[5687] := 16#D2AD;
   // UNICODE_TO_GBK[5688] := 16#564F;
   // UNICODE_TO_GBK[5689] := 16#8771;
   // UNICODE_TO_GBK[5690] := 16#5650;
   // UNICODE_TO_GBK[5691] := 16#8772;
   // UNICODE_TO_GBK[5692] := 16#5651;
   // UNICODE_TO_GBK[5693] := 16#8773;
   // UNICODE_TO_GBK[5694] := 16#5652;
   // UNICODE_TO_GBK[5695] := 16#8774;
   // UNICODE_TO_GBK[5696] := 16#5653;
   // UNICODE_TO_GBK[5697] := 16#8775;
   // UNICODE_TO_GBK[5698] := 16#5654;
   // UNICODE_TO_GBK[5699] := 16#E0E2;
   // UNICODE_TO_GBK[5700] := 16#5655;
   // UNICODE_TO_GBK[5701] := 16#8776;
   // UNICODE_TO_GBK[5702] := 16#5656;
   // UNICODE_TO_GBK[5703] := 16#8777;
   // UNICODE_TO_GBK[5704] := 16#5657;
   // UNICODE_TO_GBK[5705] := 16#E0DB;
   // UNICODE_TO_GBK[5706] := 16#5658;
   // UNICODE_TO_GBK[5707] := 16#E0D9;
   // UNICODE_TO_GBK[5708] := 16#5659;
   // UNICODE_TO_GBK[5709] := 16#E0DF;
   // UNICODE_TO_GBK[5710] := 16#565A;
   // UNICODE_TO_GBK[5711] := 16#8778;
   // UNICODE_TO_GBK[5712] := 16#565B;
   // UNICODE_TO_GBK[5713] := 16#8779;
   // UNICODE_TO_GBK[5714] := 16#565C;
   // UNICODE_TO_GBK[5715] := 16#E0E0;
   // UNICODE_TO_GBK[5716] := 16#565D;
   // UNICODE_TO_GBK[5717] := 16#877A;
   // UNICODE_TO_GBK[5718] := 16#565E;
   // UNICODE_TO_GBK[5719] := 16#877B;
   // UNICODE_TO_GBK[5720] := 16#565F;
   // UNICODE_TO_GBK[5721] := 16#877C;
   // UNICODE_TO_GBK[5722] := 16#5660;
   // UNICODE_TO_GBK[5723] := 16#877D;
   // UNICODE_TO_GBK[5724] := 16#5661;
   // UNICODE_TO_GBK[5725] := 16#877E;
   // UNICODE_TO_GBK[5726] := 16#5662;
   // UNICODE_TO_GBK[5727] := 16#E0DE;
   // UNICODE_TO_GBK[5728] := 16#5663;
   // UNICODE_TO_GBK[5729] := 16#8780;
   // UNICODE_TO_GBK[5730] := 16#5664;
   // UNICODE_TO_GBK[5731] := 16#E0E4;
   // UNICODE_TO_GBK[5732] := 16#5665;
   // UNICODE_TO_GBK[5733] := 16#8781;
   // UNICODE_TO_GBK[5734] := 16#5666;
   // UNICODE_TO_GBK[5735] := 16#8782;
   // UNICODE_TO_GBK[5736] := 16#5667;
   // UNICODE_TO_GBK[5737] := 16#8783;
   // UNICODE_TO_GBK[5738] := 16#5668;
   // UNICODE_TO_GBK[5739] := 16#C6F7;
   // UNICODE_TO_GBK[5740] := 16#5669;
   // UNICODE_TO_GBK[5741] := 16#D8AC;
   // UNICODE_TO_GBK[5742] := 16#566A;
   // UNICODE_TO_GBK[5743] := 16#D4EB;
   // UNICODE_TO_GBK[5744] := 16#566B;
   // UNICODE_TO_GBK[5745] := 16#E0E6;
   // UNICODE_TO_GBK[5746] := 16#566C;
   // UNICODE_TO_GBK[5747] := 16#CAC9;
   // UNICODE_TO_GBK[5748] := 16#566D;
   // UNICODE_TO_GBK[5749] := 16#8784;
   // UNICODE_TO_GBK[5750] := 16#566E;
   // UNICODE_TO_GBK[5751] := 16#8785;
   // UNICODE_TO_GBK[5752] := 16#566F;
   // UNICODE_TO_GBK[5753] := 16#8786;
   // UNICODE_TO_GBK[5754] := 16#5670;
   // UNICODE_TO_GBK[5755] := 16#8787;
   // UNICODE_TO_GBK[5756] := 16#5671;
   // UNICODE_TO_GBK[5757] := 16#E0E5;
   // UNICODE_TO_GBK[5758] := 16#5672;
   // UNICODE_TO_GBK[5759] := 16#8788;
   // UNICODE_TO_GBK[5760] := 16#5673;
   // UNICODE_TO_GBK[5761] := 16#8789;
   // UNICODE_TO_GBK[5762] := 16#5674;
   // UNICODE_TO_GBK[5763] := 16#878A;
   // UNICODE_TO_GBK[5764] := 16#5675;
   // UNICODE_TO_GBK[5765] := 16#878B;
   // UNICODE_TO_GBK[5766] := 16#5676;
   // UNICODE_TO_GBK[5767] := 16#B8C1;
   // UNICODE_TO_GBK[5768] := 16#5677;
   // UNICODE_TO_GBK[5769] := 16#878C;
   // UNICODE_TO_GBK[5770] := 16#5678;
   // UNICODE_TO_GBK[5771] := 16#878D;
   // UNICODE_TO_GBK[5772] := 16#5679;
   // UNICODE_TO_GBK[5773] := 16#878E;
   // UNICODE_TO_GBK[5774] := 16#567A;
   // UNICODE_TO_GBK[5775] := 16#878F;
   // UNICODE_TO_GBK[5776] := 16#567B;
   // UNICODE_TO_GBK[5777] := 16#E0E7;
   // UNICODE_TO_GBK[5778] := 16#567C;
   // UNICODE_TO_GBK[5779] := 16#E0E8;
   // UNICODE_TO_GBK[5780] := 16#567D;
   // UNICODE_TO_GBK[5781] := 16#8790;
   // UNICODE_TO_GBK[5782] := 16#567E;
   // UNICODE_TO_GBK[5783] := 16#8791;
   // UNICODE_TO_GBK[5784] := 16#567F;
   // UNICODE_TO_GBK[5785] := 16#8792;
   // UNICODE_TO_GBK[5786] := 16#5680;
   // UNICODE_TO_GBK[5787] := 16#8793;
   // UNICODE_TO_GBK[5788] := 16#5681;
   // UNICODE_TO_GBK[5789] := 16#8794;
   // UNICODE_TO_GBK[5790] := 16#5682;
   // UNICODE_TO_GBK[5791] := 16#8795;
   // UNICODE_TO_GBK[5792] := 16#5683;
   // UNICODE_TO_GBK[5793] := 16#8796;
   // UNICODE_TO_GBK[5794] := 16#5684;
   // UNICODE_TO_GBK[5795] := 16#8797;
   // UNICODE_TO_GBK[5796] := 16#5685;
   // UNICODE_TO_GBK[5797] := 16#E0E9;
   // UNICODE_TO_GBK[5798] := 16#5686;
   // UNICODE_TO_GBK[5799] := 16#E0E3;
   // UNICODE_TO_GBK[5800] := 16#5687;
   // UNICODE_TO_GBK[5801] := 16#8798;
   // UNICODE_TO_GBK[5802] := 16#5688;
   // UNICODE_TO_GBK[5803] := 16#8799;
   // UNICODE_TO_GBK[5804] := 16#5689;
   // UNICODE_TO_GBK[5805] := 16#879A;
   // UNICODE_TO_GBK[5806] := 16#568A;
   // UNICODE_TO_GBK[5807] := 16#879B;
   // UNICODE_TO_GBK[5808] := 16#568B;
   // UNICODE_TO_GBK[5809] := 16#879C;
   // UNICODE_TO_GBK[5810] := 16#568C;
   // UNICODE_TO_GBK[5811] := 16#879D;
   // UNICODE_TO_GBK[5812] := 16#568D;
   // UNICODE_TO_GBK[5813] := 16#879E;
   // UNICODE_TO_GBK[5814] := 16#568E;
   // UNICODE_TO_GBK[5815] := 16#BABF;
   // UNICODE_TO_GBK[5816] := 16#568F;
   // UNICODE_TO_GBK[5817] := 16#CCE7;
   // UNICODE_TO_GBK[5818] := 16#5690;
   // UNICODE_TO_GBK[5819] := 16#879F;
   // UNICODE_TO_GBK[5820] := 16#5691;
   // UNICODE_TO_GBK[5821] := 16#87A0;
   // UNICODE_TO_GBK[5822] := 16#5692;
   // UNICODE_TO_GBK[5823] := 16#87A1;
   // UNICODE_TO_GBK[5824] := 16#5693;
   // UNICODE_TO_GBK[5825] := 16#E0EA;
   // UNICODE_TO_GBK[5826] := 16#5694;
   // UNICODE_TO_GBK[5827] := 16#87A2;
   // UNICODE_TO_GBK[5828] := 16#5695;
   // UNICODE_TO_GBK[5829] := 16#87A3;
   // UNICODE_TO_GBK[5830] := 16#5696;
   // UNICODE_TO_GBK[5831] := 16#87A4;
   // UNICODE_TO_GBK[5832] := 16#5697;
   // UNICODE_TO_GBK[5833] := 16#87A5;
   // UNICODE_TO_GBK[5834] := 16#5698;
   // UNICODE_TO_GBK[5835] := 16#87A6;
   // UNICODE_TO_GBK[5836] := 16#5699;
   // UNICODE_TO_GBK[5837] := 16#87A7;
   // UNICODE_TO_GBK[5838] := 16#569A;
   // UNICODE_TO_GBK[5839] := 16#87A8;
   // UNICODE_TO_GBK[5840] := 16#569B;
   // UNICODE_TO_GBK[5841] := 16#87A9;
   // UNICODE_TO_GBK[5842] := 16#569C;
   // UNICODE_TO_GBK[5843] := 16#87AA;
   // UNICODE_TO_GBK[5844] := 16#569D;
   // UNICODE_TO_GBK[5845] := 16#87AB;
   // UNICODE_TO_GBK[5846] := 16#569E;
   // UNICODE_TO_GBK[5847] := 16#87AC;
   // UNICODE_TO_GBK[5848] := 16#569F;
   // UNICODE_TO_GBK[5849] := 16#87AD;
   // UNICODE_TO_GBK[5850] := 16#56A0;
   // UNICODE_TO_GBK[5851] := 16#87AE;
   // UNICODE_TO_GBK[5852] := 16#56A1;
   // UNICODE_TO_GBK[5853] := 16#87AF;
   // UNICODE_TO_GBK[5854] := 16#56A2;
   // UNICODE_TO_GBK[5855] := 16#87B0;
   // UNICODE_TO_GBK[5856] := 16#56A3;
   // UNICODE_TO_GBK[5857] := 16#CFF9;
   // UNICODE_TO_GBK[5858] := 16#56A4;
   // UNICODE_TO_GBK[5859] := 16#87B1;
   // UNICODE_TO_GBK[5860] := 16#56A5;
   // UNICODE_TO_GBK[5861] := 16#87B2;
   // UNICODE_TO_GBK[5862] := 16#56A6;
   // UNICODE_TO_GBK[5863] := 16#87B3;
   // UNICODE_TO_GBK[5864] := 16#56A7;
   // UNICODE_TO_GBK[5865] := 16#87B4;
   // UNICODE_TO_GBK[5866] := 16#56A8;
   // UNICODE_TO_GBK[5867] := 16#87B5;
   // UNICODE_TO_GBK[5868] := 16#56A9;
   // UNICODE_TO_GBK[5869] := 16#87B6;
   // UNICODE_TO_GBK[5870] := 16#56AA;
   // UNICODE_TO_GBK[5871] := 16#87B7;
   // UNICODE_TO_GBK[5872] := 16#56AB;
   // UNICODE_TO_GBK[5873] := 16#87B8;
   // UNICODE_TO_GBK[5874] := 16#56AC;
   // UNICODE_TO_GBK[5875] := 16#87B9;
   // UNICODE_TO_GBK[5876] := 16#56AD;
   // UNICODE_TO_GBK[5877] := 16#87BA;
   // UNICODE_TO_GBK[5878] := 16#56AE;
   // UNICODE_TO_GBK[5879] := 16#87BB;
   // UNICODE_TO_GBK[5880] := 16#56AF;
   // UNICODE_TO_GBK[5881] := 16#E0EB;
   // UNICODE_TO_GBK[5882] := 16#56B0;
   // UNICODE_TO_GBK[5883] := 16#87BC;
   // UNICODE_TO_GBK[5884] := 16#56B1;
   // UNICODE_TO_GBK[5885] := 16#87BD;
   // UNICODE_TO_GBK[5886] := 16#56B2;
   // UNICODE_TO_GBK[5887] := 16#87BE;
   // UNICODE_TO_GBK[5888] := 16#56B3;
   // UNICODE_TO_GBK[5889] := 16#87BF;
   // UNICODE_TO_GBK[5890] := 16#56B4;
   // UNICODE_TO_GBK[5891] := 16#87C0;
   // UNICODE_TO_GBK[5892] := 16#56B5;
   // UNICODE_TO_GBK[5893] := 16#87C1;
   // UNICODE_TO_GBK[5894] := 16#56B6;
   // UNICODE_TO_GBK[5895] := 16#87C2;
   // UNICODE_TO_GBK[5896] := 16#56B7;
   // UNICODE_TO_GBK[5897] := 16#C8C2;
   // UNICODE_TO_GBK[5898] := 16#56B8;
   // UNICODE_TO_GBK[5899] := 16#87C3;
   // UNICODE_TO_GBK[5900] := 16#56B9;
   // UNICODE_TO_GBK[5901] := 16#87C4;
   // UNICODE_TO_GBK[5902] := 16#56BA;
   // UNICODE_TO_GBK[5903] := 16#87C5;
   // UNICODE_TO_GBK[5904] := 16#56BB;
   // UNICODE_TO_GBK[5905] := 16#87C6;
   // UNICODE_TO_GBK[5906] := 16#56BC;
   // UNICODE_TO_GBK[5907] := 16#BDC0;
   // UNICODE_TO_GBK[5908] := 16#56BD;
   // UNICODE_TO_GBK[5909] := 16#87C7;
   // UNICODE_TO_GBK[5910] := 16#56BE;
   // UNICODE_TO_GBK[5911] := 16#87C8;
   // UNICODE_TO_GBK[5912] := 16#56BF;
   // UNICODE_TO_GBK[5913] := 16#87C9;
   // UNICODE_TO_GBK[5914] := 16#56C0;
   // UNICODE_TO_GBK[5915] := 16#87CA;
   // UNICODE_TO_GBK[5916] := 16#56C1;
   // UNICODE_TO_GBK[5917] := 16#87CB;
   // UNICODE_TO_GBK[5918] := 16#56C2;
   // UNICODE_TO_GBK[5919] := 16#87CC;
   // UNICODE_TO_GBK[5920] := 16#56C3;
   // UNICODE_TO_GBK[5921] := 16#87CD;
   // UNICODE_TO_GBK[5922] := 16#56C4;
   // UNICODE_TO_GBK[5923] := 16#87CE;
   // UNICODE_TO_GBK[5924] := 16#56C5;
   // UNICODE_TO_GBK[5925] := 16#87CF;
   // UNICODE_TO_GBK[5926] := 16#56C6;
   // UNICODE_TO_GBK[5927] := 16#87D0;
   // UNICODE_TO_GBK[5928] := 16#56C7;
   // UNICODE_TO_GBK[5929] := 16#87D1;
   // UNICODE_TO_GBK[5930] := 16#56C8;
   // UNICODE_TO_GBK[5931] := 16#87D2;
   // UNICODE_TO_GBK[5932] := 16#56C9;
   // UNICODE_TO_GBK[5933] := 16#87D3;
   // UNICODE_TO_GBK[5934] := 16#56CA;
   // UNICODE_TO_GBK[5935] := 16#C4D2;
   // UNICODE_TO_GBK[5936] := 16#56CB;
   // UNICODE_TO_GBK[5937] := 16#87D4;
   // UNICODE_TO_GBK[5938] := 16#56CC;
   // UNICODE_TO_GBK[5939] := 16#87D5;
   // UNICODE_TO_GBK[5940] := 16#56CD;
   // UNICODE_TO_GBK[5941] := 16#87D6;
   // UNICODE_TO_GBK[5942] := 16#56CE;
   // UNICODE_TO_GBK[5943] := 16#87D7;
   // UNICODE_TO_GBK[5944] := 16#56CF;
   // UNICODE_TO_GBK[5945] := 16#87D8;
   // UNICODE_TO_GBK[5946] := 16#56D0;
   // UNICODE_TO_GBK[5947] := 16#87D9;
   // UNICODE_TO_GBK[5948] := 16#56D1;
   // UNICODE_TO_GBK[5949] := 16#87DA;
   // UNICODE_TO_GBK[5950] := 16#56D2;
   // UNICODE_TO_GBK[5951] := 16#87DB;
   // UNICODE_TO_GBK[5952] := 16#56D3;
   // UNICODE_TO_GBK[5953] := 16#87DC;
   // UNICODE_TO_GBK[5954] := 16#56D4;
   // UNICODE_TO_GBK[5955] := 16#E0EC;
   // UNICODE_TO_GBK[5956] := 16#56D5;
   // UNICODE_TO_GBK[5957] := 16#87DD;
   // UNICODE_TO_GBK[5958] := 16#56D6;
   // UNICODE_TO_GBK[5959] := 16#87DE;
   // UNICODE_TO_GBK[5960] := 16#56D7;
   // UNICODE_TO_GBK[5961] := 16#E0ED;
   // UNICODE_TO_GBK[5962] := 16#56D8;
   // UNICODE_TO_GBK[5963] := 16#87DF;
   // UNICODE_TO_GBK[5964] := 16#56D9;
   // UNICODE_TO_GBK[5965] := 16#87E0;
   // UNICODE_TO_GBK[5966] := 16#56DA;
   // UNICODE_TO_GBK[5967] := 16#C7F4;
   // UNICODE_TO_GBK[5968] := 16#56DB;
   // UNICODE_TO_GBK[5969] := 16#CBC4;
   // UNICODE_TO_GBK[5970] := 16#56DC;
   // UNICODE_TO_GBK[5971] := 16#87E1;
   // UNICODE_TO_GBK[5972] := 16#56DD;
   // UNICODE_TO_GBK[5973] := 16#E0EE;
   // UNICODE_TO_GBK[5974] := 16#56DE;
   // UNICODE_TO_GBK[5975] := 16#BBD8;
   // UNICODE_TO_GBK[5976] := 16#56DF;
   // UNICODE_TO_GBK[5977] := 16#D8B6;
   // UNICODE_TO_GBK[5978] := 16#56E0;
   // UNICODE_TO_GBK[5979] := 16#D2F2;
   // UNICODE_TO_GBK[5980] := 16#56E1;
   // UNICODE_TO_GBK[5981] := 16#E0EF;
   // UNICODE_TO_GBK[5982] := 16#56E2;
   // UNICODE_TO_GBK[5983] := 16#CDC5;
   // UNICODE_TO_GBK[5984] := 16#56E3;
   // UNICODE_TO_GBK[5985] := 16#87E2;
   // UNICODE_TO_GBK[5986] := 16#56E4;
   // UNICODE_TO_GBK[5987] := 16#B6DA;
   // UNICODE_TO_GBK[5988] := 16#56E5;
   // UNICODE_TO_GBK[5989] := 16#87E3;
   // UNICODE_TO_GBK[5990] := 16#56E6;
   // UNICODE_TO_GBK[5991] := 16#87E4;
   // UNICODE_TO_GBK[5992] := 16#56E7;
   // UNICODE_TO_GBK[5993] := 16#87E5;
   // UNICODE_TO_GBK[5994] := 16#56E8;
   // UNICODE_TO_GBK[5995] := 16#87E6;
   // UNICODE_TO_GBK[5996] := 16#56E9;
   // UNICODE_TO_GBK[5997] := 16#87E7;
   // UNICODE_TO_GBK[5998] := 16#56EA;
   // UNICODE_TO_GBK[5999] := 16#87E8;
   // UNICODE_TO_GBK[6000] := 16#56EB;
   // UNICODE_TO_GBK[6001] := 16#E0F1;
   // UNICODE_TO_GBK[6002] := 16#56EC;
   // UNICODE_TO_GBK[6003] := 16#87E9;
   // UNICODE_TO_GBK[6004] := 16#56ED;
   // UNICODE_TO_GBK[6005] := 16#D4B0;
   // UNICODE_TO_GBK[6006] := 16#56EE;
   // UNICODE_TO_GBK[6007] := 16#87EA;
   // UNICODE_TO_GBK[6008] := 16#56EF;
   // UNICODE_TO_GBK[6009] := 16#87EB;
   // UNICODE_TO_GBK[6010] := 16#56F0;
   // UNICODE_TO_GBK[6011] := 16#C0A7;
   // UNICODE_TO_GBK[6012] := 16#56F1;
   // UNICODE_TO_GBK[6013] := 16#B4D1;
   // UNICODE_TO_GBK[6014] := 16#56F2;
   // UNICODE_TO_GBK[6015] := 16#87EC;
   // UNICODE_TO_GBK[6016] := 16#56F3;
   // UNICODE_TO_GBK[6017] := 16#87ED;
   // UNICODE_TO_GBK[6018] := 16#56F4;
   // UNICODE_TO_GBK[6019] := 16#CEA7;
   // UNICODE_TO_GBK[6020] := 16#56F5;
   // UNICODE_TO_GBK[6021] := 16#E0F0;
   // UNICODE_TO_GBK[6022] := 16#56F6;
   // UNICODE_TO_GBK[6023] := 16#87EE;
   // UNICODE_TO_GBK[6024] := 16#56F7;
   // UNICODE_TO_GBK[6025] := 16#87EF;
   // UNICODE_TO_GBK[6026] := 16#56F8;
   // UNICODE_TO_GBK[6027] := 16#87F0;
   // UNICODE_TO_GBK[6028] := 16#56F9;
   // UNICODE_TO_GBK[6029] := 16#E0F2;
   // UNICODE_TO_GBK[6030] := 16#56FA;
   // UNICODE_TO_GBK[6031] := 16#B9CC;
   // UNICODE_TO_GBK[6032] := 16#56FB;
   // UNICODE_TO_GBK[6033] := 16#87F1;
   // UNICODE_TO_GBK[6034] := 16#56FC;
   // UNICODE_TO_GBK[6035] := 16#87F2;
   // UNICODE_TO_GBK[6036] := 16#56FD;
   // UNICODE_TO_GBK[6037] := 16#B9FA;
   // UNICODE_TO_GBK[6038] := 16#56FE;
   // UNICODE_TO_GBK[6039] := 16#CDBC;
   // UNICODE_TO_GBK[6040] := 16#56FF;
   // UNICODE_TO_GBK[6041] := 16#E0F3;
   // UNICODE_TO_GBK[6042] := 16#5700;
   // UNICODE_TO_GBK[6043] := 16#87F3;
   // UNICODE_TO_GBK[6044] := 16#5701;
   // UNICODE_TO_GBK[6045] := 16#87F4;
   // UNICODE_TO_GBK[6046] := 16#5702;
   // UNICODE_TO_GBK[6047] := 16#87F5;
   // UNICODE_TO_GBK[6048] := 16#5703;
   // UNICODE_TO_GBK[6049] := 16#C6D4;
   // UNICODE_TO_GBK[6050] := 16#5704;
   // UNICODE_TO_GBK[6051] := 16#E0F4;
   // UNICODE_TO_GBK[6052] := 16#5705;
   // UNICODE_TO_GBK[6053] := 16#87F6;
   // UNICODE_TO_GBK[6054] := 16#5706;
   // UNICODE_TO_GBK[6055] := 16#D4B2;
   // UNICODE_TO_GBK[6056] := 16#5707;
   // UNICODE_TO_GBK[6057] := 16#87F7;
   // UNICODE_TO_GBK[6058] := 16#5708;
   // UNICODE_TO_GBK[6059] := 16#C8A6;
   // UNICODE_TO_GBK[6060] := 16#5709;
   // UNICODE_TO_GBK[6061] := 16#E0F6;
   // UNICODE_TO_GBK[6062] := 16#570A;
   // UNICODE_TO_GBK[6063] := 16#E0F5;
   // UNICODE_TO_GBK[6064] := 16#570B;
   // UNICODE_TO_GBK[6065] := 16#87F8;
   // UNICODE_TO_GBK[6066] := 16#570C;
   // UNICODE_TO_GBK[6067] := 16#87F9;
   // UNICODE_TO_GBK[6068] := 16#570D;
   // UNICODE_TO_GBK[6069] := 16#87FA;
   // UNICODE_TO_GBK[6070] := 16#570E;
   // UNICODE_TO_GBK[6071] := 16#87FB;
   // UNICODE_TO_GBK[6072] := 16#570F;
   // UNICODE_TO_GBK[6073] := 16#87FC;
   // UNICODE_TO_GBK[6074] := 16#5710;
   // UNICODE_TO_GBK[6075] := 16#87FD;
   // UNICODE_TO_GBK[6076] := 16#5711;
   // UNICODE_TO_GBK[6077] := 16#87FE;
   // UNICODE_TO_GBK[6078] := 16#5712;
   // UNICODE_TO_GBK[6079] := 16#8840;
   // UNICODE_TO_GBK[6080] := 16#5713;
   // UNICODE_TO_GBK[6081] := 16#8841;
   // UNICODE_TO_GBK[6082] := 16#5714;
   // UNICODE_TO_GBK[6083] := 16#8842;
   // UNICODE_TO_GBK[6084] := 16#5715;
   // UNICODE_TO_GBK[6085] := 16#8843;
   // UNICODE_TO_GBK[6086] := 16#5716;
   // UNICODE_TO_GBK[6087] := 16#8844;
   // UNICODE_TO_GBK[6088] := 16#5717;
   // UNICODE_TO_GBK[6089] := 16#8845;
   // UNICODE_TO_GBK[6090] := 16#5718;
   // UNICODE_TO_GBK[6091] := 16#8846;
   // UNICODE_TO_GBK[6092] := 16#5719;
   // UNICODE_TO_GBK[6093] := 16#8847;
   // UNICODE_TO_GBK[6094] := 16#571A;
   // UNICODE_TO_GBK[6095] := 16#8848;
   // UNICODE_TO_GBK[6096] := 16#571B;
   // UNICODE_TO_GBK[6097] := 16#8849;
   // UNICODE_TO_GBK[6098] := 16#571C;
   // UNICODE_TO_GBK[6099] := 16#E0F7;
   // UNICODE_TO_GBK[6100] := 16#571D;
   // UNICODE_TO_GBK[6101] := 16#884A;
   // UNICODE_TO_GBK[6102] := 16#571E;
   // UNICODE_TO_GBK[6103] := 16#884B;
   // UNICODE_TO_GBK[6104] := 16#571F;
   // UNICODE_TO_GBK[6105] := 16#CDC1;
   // UNICODE_TO_GBK[6106] := 16#5720;
   // UNICODE_TO_GBK[6107] := 16#884C;
   // UNICODE_TO_GBK[6108] := 16#5721;
   // UNICODE_TO_GBK[6109] := 16#884D;
   // UNICODE_TO_GBK[6110] := 16#5722;
   // UNICODE_TO_GBK[6111] := 16#884E;
   // UNICODE_TO_GBK[6112] := 16#5723;
   // UNICODE_TO_GBK[6113] := 16#CAA5;
   // UNICODE_TO_GBK[6114] := 16#5724;
   // UNICODE_TO_GBK[6115] := 16#884F;
   // UNICODE_TO_GBK[6116] := 16#5725;
   // UNICODE_TO_GBK[6117] := 16#8850;
   // UNICODE_TO_GBK[6118] := 16#5726;
   // UNICODE_TO_GBK[6119] := 16#8851;
   // UNICODE_TO_GBK[6120] := 16#5727;
   // UNICODE_TO_GBK[6121] := 16#8852;
   // UNICODE_TO_GBK[6122] := 16#5728;
   // UNICODE_TO_GBK[6123] := 16#D4DA;
   // UNICODE_TO_GBK[6124] := 16#5729;
   // UNICODE_TO_GBK[6125] := 16#DBD7;
   // UNICODE_TO_GBK[6126] := 16#572A;
   // UNICODE_TO_GBK[6127] := 16#DBD9;
   // UNICODE_TO_GBK[6128] := 16#572B;
   // UNICODE_TO_GBK[6129] := 16#8853;
   // UNICODE_TO_GBK[6130] := 16#572C;
   // UNICODE_TO_GBK[6131] := 16#DBD8;
   // UNICODE_TO_GBK[6132] := 16#572D;
   // UNICODE_TO_GBK[6133] := 16#B9E7;
   // UNICODE_TO_GBK[6134] := 16#572E;
   // UNICODE_TO_GBK[6135] := 16#DBDC;
   // UNICODE_TO_GBK[6136] := 16#572F;
   // UNICODE_TO_GBK[6137] := 16#DBDD;
   // UNICODE_TO_GBK[6138] := 16#5730;
   // UNICODE_TO_GBK[6139] := 16#B5D8;
   // UNICODE_TO_GBK[6140] := 16#5731;
   // UNICODE_TO_GBK[6141] := 16#8854;
   // UNICODE_TO_GBK[6142] := 16#5732;
   // UNICODE_TO_GBK[6143] := 16#8855;
   // UNICODE_TO_GBK[6144] := 16#5733;
   // UNICODE_TO_GBK[6145] := 16#DBDA;
   // UNICODE_TO_GBK[6146] := 16#5734;
   // UNICODE_TO_GBK[6147] := 16#8856;
   // UNICODE_TO_GBK[6148] := 16#5735;
   // UNICODE_TO_GBK[6149] := 16#8857;
   // UNICODE_TO_GBK[6150] := 16#5736;
   // UNICODE_TO_GBK[6151] := 16#8858;
   // UNICODE_TO_GBK[6152] := 16#5737;
   // UNICODE_TO_GBK[6153] := 16#8859;
   // UNICODE_TO_GBK[6154] := 16#5738;
   // UNICODE_TO_GBK[6155] := 16#885A;
   // UNICODE_TO_GBK[6156] := 16#5739;
   // UNICODE_TO_GBK[6157] := 16#DBDB;
   // UNICODE_TO_GBK[6158] := 16#573A;
   // UNICODE_TO_GBK[6159] := 16#B3A1;
   // UNICODE_TO_GBK[6160] := 16#573B;
   // UNICODE_TO_GBK[6161] := 16#DBDF;
   // UNICODE_TO_GBK[6162] := 16#573C;
   // UNICODE_TO_GBK[6163] := 16#885B;
   // UNICODE_TO_GBK[6164] := 16#573D;
   // UNICODE_TO_GBK[6165] := 16#885C;
   // UNICODE_TO_GBK[6166] := 16#573E;
   // UNICODE_TO_GBK[6167] := 16#BBF8;
   // UNICODE_TO_GBK[6168] := 16#573F;
   // UNICODE_TO_GBK[6169] := 16#885D;
   // UNICODE_TO_GBK[6170] := 16#5740;
   // UNICODE_TO_GBK[6171] := 16#D6B7;
   // UNICODE_TO_GBK[6172] := 16#5741;
   // UNICODE_TO_GBK[6173] := 16#885E;
   // UNICODE_TO_GBK[6174] := 16#5742;
   // UNICODE_TO_GBK[6175] := 16#DBE0;
   // UNICODE_TO_GBK[6176] := 16#5743;
   // UNICODE_TO_GBK[6177] := 16#885F;
   // UNICODE_TO_GBK[6178] := 16#5744;
   // UNICODE_TO_GBK[6179] := 16#8860;
   // UNICODE_TO_GBK[6180] := 16#5745;
   // UNICODE_TO_GBK[6181] := 16#8861;
   // UNICODE_TO_GBK[6182] := 16#5746;
   // UNICODE_TO_GBK[6183] := 16#8862;
   // UNICODE_TO_GBK[6184] := 16#5747;
   // UNICODE_TO_GBK[6185] := 16#BEF9;
   // UNICODE_TO_GBK[6186] := 16#5748;
   // UNICODE_TO_GBK[6187] := 16#8863;
   // UNICODE_TO_GBK[6188] := 16#5749;
   // UNICODE_TO_GBK[6189] := 16#8864;
   // UNICODE_TO_GBK[6190] := 16#574A;
   // UNICODE_TO_GBK[6191] := 16#B7BB;
   // UNICODE_TO_GBK[6192] := 16#574B;
   // UNICODE_TO_GBK[6193] := 16#8865;
   // UNICODE_TO_GBK[6194] := 16#574C;
   // UNICODE_TO_GBK[6195] := 16#DBD0;
   // UNICODE_TO_GBK[6196] := 16#574D;
   // UNICODE_TO_GBK[6197] := 16#CCAE;
   // UNICODE_TO_GBK[6198] := 16#574E;
   // UNICODE_TO_GBK[6199] := 16#BFB2;
   // UNICODE_TO_GBK[6200] := 16#574F;
   // UNICODE_TO_GBK[6201] := 16#BBB5;
   // UNICODE_TO_GBK[6202] := 16#5750;
   // UNICODE_TO_GBK[6203] := 16#D7F8;
   // UNICODE_TO_GBK[6204] := 16#5751;
   // UNICODE_TO_GBK[6205] := 16#BFD3;
   // UNICODE_TO_GBK[6206] := 16#5752;
   // UNICODE_TO_GBK[6207] := 16#8866;
   // UNICODE_TO_GBK[6208] := 16#5753;
   // UNICODE_TO_GBK[6209] := 16#8867;
   // UNICODE_TO_GBK[6210] := 16#5754;
   // UNICODE_TO_GBK[6211] := 16#8868;
   // UNICODE_TO_GBK[6212] := 16#5755;
   // UNICODE_TO_GBK[6213] := 16#8869;
   // UNICODE_TO_GBK[6214] := 16#5756;
   // UNICODE_TO_GBK[6215] := 16#886A;
   // UNICODE_TO_GBK[6216] := 16#5757;
   // UNICODE_TO_GBK[6217] := 16#BFE9;
   // UNICODE_TO_GBK[6218] := 16#5758;
   // UNICODE_TO_GBK[6219] := 16#886B;
   // UNICODE_TO_GBK[6220] := 16#5759;
   // UNICODE_TO_GBK[6221] := 16#886C;
   // UNICODE_TO_GBK[6222] := 16#575A;
   // UNICODE_TO_GBK[6223] := 16#BCE1;
   // UNICODE_TO_GBK[6224] := 16#575B;
   // UNICODE_TO_GBK[6225] := 16#CCB3;
   // UNICODE_TO_GBK[6226] := 16#575C;
   // UNICODE_TO_GBK[6227] := 16#DBDE;
   // UNICODE_TO_GBK[6228] := 16#575D;
   // UNICODE_TO_GBK[6229] := 16#B0D3;
   // UNICODE_TO_GBK[6230] := 16#575E;
   // UNICODE_TO_GBK[6231] := 16#CEEB;
   // UNICODE_TO_GBK[6232] := 16#575F;
   // UNICODE_TO_GBK[6233] := 16#B7D8;
   // UNICODE_TO_GBK[6234] := 16#5760;
   // UNICODE_TO_GBK[6235] := 16#D7B9;
   // UNICODE_TO_GBK[6236] := 16#5761;
   // UNICODE_TO_GBK[6237] := 16#C6C2;
   // UNICODE_TO_GBK[6238] := 16#5762;
   // UNICODE_TO_GBK[6239] := 16#886D;
   // UNICODE_TO_GBK[6240] := 16#5763;
   // UNICODE_TO_GBK[6241] := 16#886E;
   // UNICODE_TO_GBK[6242] := 16#5764;
   // UNICODE_TO_GBK[6243] := 16#C0A4;
   // UNICODE_TO_GBK[6244] := 16#5765;
   // UNICODE_TO_GBK[6245] := 16#886F;
   // UNICODE_TO_GBK[6246] := 16#5766;
   // UNICODE_TO_GBK[6247] := 16#CCB9;
   // UNICODE_TO_GBK[6248] := 16#5767;
   // UNICODE_TO_GBK[6249] := 16#8870;
   // UNICODE_TO_GBK[6250] := 16#5768;
   // UNICODE_TO_GBK[6251] := 16#DBE7;
   // UNICODE_TO_GBK[6252] := 16#5769;
   // UNICODE_TO_GBK[6253] := 16#DBE1;
   // UNICODE_TO_GBK[6254] := 16#576A;
   // UNICODE_TO_GBK[6255] := 16#C6BA;
   // UNICODE_TO_GBK[6256] := 16#576B;
   // UNICODE_TO_GBK[6257] := 16#DBE3;
   // UNICODE_TO_GBK[6258] := 16#576C;
   // UNICODE_TO_GBK[6259] := 16#8871;
   // UNICODE_TO_GBK[6260] := 16#576D;
   // UNICODE_TO_GBK[6261] := 16#DBE8;
   // UNICODE_TO_GBK[6262] := 16#576E;
   // UNICODE_TO_GBK[6263] := 16#8872;
   // UNICODE_TO_GBK[6264] := 16#576F;
   // UNICODE_TO_GBK[6265] := 16#C5F7;
   // UNICODE_TO_GBK[6266] := 16#5770;
   // UNICODE_TO_GBK[6267] := 16#8873;
   // UNICODE_TO_GBK[6268] := 16#5771;
   // UNICODE_TO_GBK[6269] := 16#8874;
   // UNICODE_TO_GBK[6270] := 16#5772;
   // UNICODE_TO_GBK[6271] := 16#8875;
   // UNICODE_TO_GBK[6272] := 16#5773;
   // UNICODE_TO_GBK[6273] := 16#DBEA;
   // UNICODE_TO_GBK[6274] := 16#5774;
   // UNICODE_TO_GBK[6275] := 16#8876;
   // UNICODE_TO_GBK[6276] := 16#5775;
   // UNICODE_TO_GBK[6277] := 16#8877;
   // UNICODE_TO_GBK[6278] := 16#5776;
   // UNICODE_TO_GBK[6279] := 16#DBE9;
   // UNICODE_TO_GBK[6280] := 16#5777;
   // UNICODE_TO_GBK[6281] := 16#BFC0;
   // UNICODE_TO_GBK[6282] := 16#5778;
   // UNICODE_TO_GBK[6283] := 16#8878;
   // UNICODE_TO_GBK[6284] := 16#5779;
   // UNICODE_TO_GBK[6285] := 16#8879;
   // UNICODE_TO_GBK[6286] := 16#577A;
   // UNICODE_TO_GBK[6287] := 16#887A;
   // UNICODE_TO_GBK[6288] := 16#577B;
   // UNICODE_TO_GBK[6289] := 16#DBE6;
   // UNICODE_TO_GBK[6290] := 16#577C;
   // UNICODE_TO_GBK[6291] := 16#DBE5;
   // UNICODE_TO_GBK[6292] := 16#577D;
   // UNICODE_TO_GBK[6293] := 16#887B;
   // UNICODE_TO_GBK[6294] := 16#577E;
   // UNICODE_TO_GBK[6295] := 16#887C;
   // UNICODE_TO_GBK[6296] := 16#577F;
   // UNICODE_TO_GBK[6297] := 16#887D;
   // UNICODE_TO_GBK[6298] := 16#5780;
   // UNICODE_TO_GBK[6299] := 16#887E;
   // UNICODE_TO_GBK[6300] := 16#5781;
   // UNICODE_TO_GBK[6301] := 16#8880;
   // UNICODE_TO_GBK[6302] := 16#5782;
   // UNICODE_TO_GBK[6303] := 16#B4B9;
   // UNICODE_TO_GBK[6304] := 16#5783;
   // UNICODE_TO_GBK[6305] := 16#C0AC;
   // UNICODE_TO_GBK[6306] := 16#5784;
   // UNICODE_TO_GBK[6307] := 16#C2A2;
   // UNICODE_TO_GBK[6308] := 16#5785;
   // UNICODE_TO_GBK[6309] := 16#DBE2;
   // UNICODE_TO_GBK[6310] := 16#5786;
   // UNICODE_TO_GBK[6311] := 16#DBE4;
   // UNICODE_TO_GBK[6312] := 16#5787;
   // UNICODE_TO_GBK[6313] := 16#8881;
   // UNICODE_TO_GBK[6314] := 16#5788;
   // UNICODE_TO_GBK[6315] := 16#8882;
   // UNICODE_TO_GBK[6316] := 16#5789;
   // UNICODE_TO_GBK[6317] := 16#8883;
   // UNICODE_TO_GBK[6318] := 16#578A;
   // UNICODE_TO_GBK[6319] := 16#8884;
   // UNICODE_TO_GBK[6320] := 16#578B;
   // UNICODE_TO_GBK[6321] := 16#D0CD;
   // UNICODE_TO_GBK[6322] := 16#578C;
   // UNICODE_TO_GBK[6323] := 16#DBED;
   // UNICODE_TO_GBK[6324] := 16#578D;
   // UNICODE_TO_GBK[6325] := 16#8885;
   // UNICODE_TO_GBK[6326] := 16#578E;
   // UNICODE_TO_GBK[6327] := 16#8886;
   // UNICODE_TO_GBK[6328] := 16#578F;
   // UNICODE_TO_GBK[6329] := 16#8887;
   // UNICODE_TO_GBK[6330] := 16#5790;
   // UNICODE_TO_GBK[6331] := 16#8888;
   // UNICODE_TO_GBK[6332] := 16#5791;
   // UNICODE_TO_GBK[6333] := 16#8889;
   // UNICODE_TO_GBK[6334] := 16#5792;
   // UNICODE_TO_GBK[6335] := 16#C0DD;
   // UNICODE_TO_GBK[6336] := 16#5793;
   // UNICODE_TO_GBK[6337] := 16#DBF2;
   // UNICODE_TO_GBK[6338] := 16#5794;
   // UNICODE_TO_GBK[6339] := 16#888A;
   // UNICODE_TO_GBK[6340] := 16#5795;
   // UNICODE_TO_GBK[6341] := 16#888B;
   // UNICODE_TO_GBK[6342] := 16#5796;
   // UNICODE_TO_GBK[6343] := 16#888C;
   // UNICODE_TO_GBK[6344] := 16#5797;
   // UNICODE_TO_GBK[6345] := 16#888D;
   // UNICODE_TO_GBK[6346] := 16#5798;
   // UNICODE_TO_GBK[6347] := 16#888E;
   // UNICODE_TO_GBK[6348] := 16#5799;
   // UNICODE_TO_GBK[6349] := 16#888F;
   // UNICODE_TO_GBK[6350] := 16#579A;
   // UNICODE_TO_GBK[6351] := 16#8890;
   // UNICODE_TO_GBK[6352] := 16#579B;
   // UNICODE_TO_GBK[6353] := 16#B6E2;
   // UNICODE_TO_GBK[6354] := 16#579C;
   // UNICODE_TO_GBK[6355] := 16#8891;
   // UNICODE_TO_GBK[6356] := 16#579D;
   // UNICODE_TO_GBK[6357] := 16#8892;
   // UNICODE_TO_GBK[6358] := 16#579E;
   // UNICODE_TO_GBK[6359] := 16#8893;
   // UNICODE_TO_GBK[6360] := 16#579F;
   // UNICODE_TO_GBK[6361] := 16#8894;
   // UNICODE_TO_GBK[6362] := 16#57A0;
   // UNICODE_TO_GBK[6363] := 16#DBF3;
   // UNICODE_TO_GBK[6364] := 16#57A1;
   // UNICODE_TO_GBK[6365] := 16#DBD2;
   // UNICODE_TO_GBK[6366] := 16#57A2;
   // UNICODE_TO_GBK[6367] := 16#B9B8;
   // UNICODE_TO_GBK[6368] := 16#57A3;
   // UNICODE_TO_GBK[6369] := 16#D4AB;
   // UNICODE_TO_GBK[6370] := 16#57A4;
   // UNICODE_TO_GBK[6371] := 16#DBEC;
   // UNICODE_TO_GBK[6372] := 16#57A5;
   // UNICODE_TO_GBK[6373] := 16#8895;
   // UNICODE_TO_GBK[6374] := 16#57A6;
   // UNICODE_TO_GBK[6375] := 16#BFD1;
   // UNICODE_TO_GBK[6376] := 16#57A7;
   // UNICODE_TO_GBK[6377] := 16#DBF0;
   // UNICODE_TO_GBK[6378] := 16#57A8;
   // UNICODE_TO_GBK[6379] := 16#8896;
   // UNICODE_TO_GBK[6380] := 16#57A9;
   // UNICODE_TO_GBK[6381] := 16#DBD1;
   // UNICODE_TO_GBK[6382] := 16#57AA;
   // UNICODE_TO_GBK[6383] := 16#8897;
   // UNICODE_TO_GBK[6384] := 16#57AB;
   // UNICODE_TO_GBK[6385] := 16#B5E6;
   // UNICODE_TO_GBK[6386] := 16#57AC;
   // UNICODE_TO_GBK[6387] := 16#8898;
   // UNICODE_TO_GBK[6388] := 16#57AD;
   // UNICODE_TO_GBK[6389] := 16#DBEB;
   // UNICODE_TO_GBK[6390] := 16#57AE;
   // UNICODE_TO_GBK[6391] := 16#BFE5;
   // UNICODE_TO_GBK[6392] := 16#57AF;
   // UNICODE_TO_GBK[6393] := 16#8899;
   // UNICODE_TO_GBK[6394] := 16#57B0;
   // UNICODE_TO_GBK[6395] := 16#889A;
   // UNICODE_TO_GBK[6396] := 16#57B1;
   // UNICODE_TO_GBK[6397] := 16#889B;
   // UNICODE_TO_GBK[6398] := 16#57B2;
   // UNICODE_TO_GBK[6399] := 16#DBEE;
   // UNICODE_TO_GBK[6400] := 16#57B3;
   // UNICODE_TO_GBK[6401] := 16#889C;
   // UNICODE_TO_GBK[6402] := 16#57B4;
   // UNICODE_TO_GBK[6403] := 16#DBF1;
   // UNICODE_TO_GBK[6404] := 16#57B5;
   // UNICODE_TO_GBK[6405] := 16#889D;
   // UNICODE_TO_GBK[6406] := 16#57B6;
   // UNICODE_TO_GBK[6407] := 16#889E;
   // UNICODE_TO_GBK[6408] := 16#57B7;
   // UNICODE_TO_GBK[6409] := 16#889F;
   // UNICODE_TO_GBK[6410] := 16#57B8;
   // UNICODE_TO_GBK[6411] := 16#DBF9;
   // UNICODE_TO_GBK[6412] := 16#57B9;
   // UNICODE_TO_GBK[6413] := 16#88A0;
   // UNICODE_TO_GBK[6414] := 16#57BA;
   // UNICODE_TO_GBK[6415] := 16#88A1;
   // UNICODE_TO_GBK[6416] := 16#57BB;
   // UNICODE_TO_GBK[6417] := 16#88A2;
   // UNICODE_TO_GBK[6418] := 16#57BC;
   // UNICODE_TO_GBK[6419] := 16#88A3;
   // UNICODE_TO_GBK[6420] := 16#57BD;
   // UNICODE_TO_GBK[6421] := 16#88A4;
   // UNICODE_TO_GBK[6422] := 16#57BE;
   // UNICODE_TO_GBK[6423] := 16#88A5;
   // UNICODE_TO_GBK[6424] := 16#57BF;
   // UNICODE_TO_GBK[6425] := 16#88A6;
   // UNICODE_TO_GBK[6426] := 16#57C0;
   // UNICODE_TO_GBK[6427] := 16#88A7;
   // UNICODE_TO_GBK[6428] := 16#57C1;
   // UNICODE_TO_GBK[6429] := 16#88A8;
   // UNICODE_TO_GBK[6430] := 16#57C2;
   // UNICODE_TO_GBK[6431] := 16#B9A1;
   // UNICODE_TO_GBK[6432] := 16#57C3;
   // UNICODE_TO_GBK[6433] := 16#B0A3;
   // UNICODE_TO_GBK[6434] := 16#57C4;
   // UNICODE_TO_GBK[6435] := 16#88A9;
   // UNICODE_TO_GBK[6436] := 16#57C5;
   // UNICODE_TO_GBK[6437] := 16#88AA;
   // UNICODE_TO_GBK[6438] := 16#57C6;
   // UNICODE_TO_GBK[6439] := 16#88AB;
   // UNICODE_TO_GBK[6440] := 16#57C7;
   // UNICODE_TO_GBK[6441] := 16#88AC;
   // UNICODE_TO_GBK[6442] := 16#57C8;
   // UNICODE_TO_GBK[6443] := 16#88AD;
   // UNICODE_TO_GBK[6444] := 16#57C9;
   // UNICODE_TO_GBK[6445] := 16#88AE;
   // UNICODE_TO_GBK[6446] := 16#57CA;
   // UNICODE_TO_GBK[6447] := 16#88AF;
   // UNICODE_TO_GBK[6448] := 16#57CB;
   // UNICODE_TO_GBK[6449] := 16#C2F1;
   // UNICODE_TO_GBK[6450] := 16#57CC;
   // UNICODE_TO_GBK[6451] := 16#88B0;
   // UNICODE_TO_GBK[6452] := 16#57CD;
   // UNICODE_TO_GBK[6453] := 16#88B1;
   // UNICODE_TO_GBK[6454] := 16#57CE;
   // UNICODE_TO_GBK[6455] := 16#B3C7;
   // UNICODE_TO_GBK[6456] := 16#57CF;
   // UNICODE_TO_GBK[6457] := 16#DBEF;
   // UNICODE_TO_GBK[6458] := 16#57D0;
   // UNICODE_TO_GBK[6459] := 16#88B2;
   // UNICODE_TO_GBK[6460] := 16#57D1;
   // UNICODE_TO_GBK[6461] := 16#88B3;
   // UNICODE_TO_GBK[6462] := 16#57D2;
   // UNICODE_TO_GBK[6463] := 16#DBF8;
   // UNICODE_TO_GBK[6464] := 16#57D3;
   // UNICODE_TO_GBK[6465] := 16#88B4;
   // UNICODE_TO_GBK[6466] := 16#57D4;
   // UNICODE_TO_GBK[6467] := 16#C6D2;
   // UNICODE_TO_GBK[6468] := 16#57D5;
   // UNICODE_TO_GBK[6469] := 16#DBF4;
   // UNICODE_TO_GBK[6470] := 16#57D6;
   // UNICODE_TO_GBK[6471] := 16#88B5;
   // UNICODE_TO_GBK[6472] := 16#57D7;
   // UNICODE_TO_GBK[6473] := 16#88B6;
   // UNICODE_TO_GBK[6474] := 16#57D8;
   // UNICODE_TO_GBK[6475] := 16#DBF5;
   // UNICODE_TO_GBK[6476] := 16#57D9;
   // UNICODE_TO_GBK[6477] := 16#DBF7;
   // UNICODE_TO_GBK[6478] := 16#57DA;
   // UNICODE_TO_GBK[6479] := 16#DBF6;
   // UNICODE_TO_GBK[6480] := 16#57DB;
   // UNICODE_TO_GBK[6481] := 16#88B7;
   // UNICODE_TO_GBK[6482] := 16#57DC;
   // UNICODE_TO_GBK[6483] := 16#88B8;
   // UNICODE_TO_GBK[6484] := 16#57DD;
   // UNICODE_TO_GBK[6485] := 16#DBFE;
   // UNICODE_TO_GBK[6486] := 16#57DE;
   // UNICODE_TO_GBK[6487] := 16#88B9;
   // UNICODE_TO_GBK[6488] := 16#57DF;
   // UNICODE_TO_GBK[6489] := 16#D3F2;
   // UNICODE_TO_GBK[6490] := 16#57E0;
   // UNICODE_TO_GBK[6491] := 16#B2BA;
   // UNICODE_TO_GBK[6492] := 16#57E1;
   // UNICODE_TO_GBK[6493] := 16#88BA;
   // UNICODE_TO_GBK[6494] := 16#57E2;
   // UNICODE_TO_GBK[6495] := 16#88BB;
   // UNICODE_TO_GBK[6496] := 16#57E3;
   // UNICODE_TO_GBK[6497] := 16#88BC;
   // UNICODE_TO_GBK[6498] := 16#57E4;
   // UNICODE_TO_GBK[6499] := 16#DBFD;
   // UNICODE_TO_GBK[6500] := 16#57E5;
   // UNICODE_TO_GBK[6501] := 16#88BD;
   // UNICODE_TO_GBK[6502] := 16#57E6;
   // UNICODE_TO_GBK[6503] := 16#88BE;
   // UNICODE_TO_GBK[6504] := 16#57E7;
   // UNICODE_TO_GBK[6505] := 16#88BF;
   // UNICODE_TO_GBK[6506] := 16#57E8;
   // UNICODE_TO_GBK[6507] := 16#88C0;
   // UNICODE_TO_GBK[6508] := 16#57E9;
   // UNICODE_TO_GBK[6509] := 16#88C1;
   // UNICODE_TO_GBK[6510] := 16#57EA;
   // UNICODE_TO_GBK[6511] := 16#88C2;
   // UNICODE_TO_GBK[6512] := 16#57EB;
   // UNICODE_TO_GBK[6513] := 16#88C3;
   // UNICODE_TO_GBK[6514] := 16#57EC;
   // UNICODE_TO_GBK[6515] := 16#88C4;
   // UNICODE_TO_GBK[6516] := 16#57ED;
   // UNICODE_TO_GBK[6517] := 16#DCA4;
   // UNICODE_TO_GBK[6518] := 16#57EE;
   // UNICODE_TO_GBK[6519] := 16#88C5;
   // UNICODE_TO_GBK[6520] := 16#57EF;
   // UNICODE_TO_GBK[6521] := 16#DBFB;
   // UNICODE_TO_GBK[6522] := 16#57F0;
   // UNICODE_TO_GBK[6523] := 16#88C6;
   // UNICODE_TO_GBK[6524] := 16#57F1;
   // UNICODE_TO_GBK[6525] := 16#88C7;
   // UNICODE_TO_GBK[6526] := 16#57F2;
   // UNICODE_TO_GBK[6527] := 16#88C8;
   // UNICODE_TO_GBK[6528] := 16#57F3;
   // UNICODE_TO_GBK[6529] := 16#88C9;
   // UNICODE_TO_GBK[6530] := 16#57F4;
   // UNICODE_TO_GBK[6531] := 16#DBFA;
   // UNICODE_TO_GBK[6532] := 16#57F5;
   // UNICODE_TO_GBK[6533] := 16#88CA;
   // UNICODE_TO_GBK[6534] := 16#57F6;
   // UNICODE_TO_GBK[6535] := 16#88CB;
   // UNICODE_TO_GBK[6536] := 16#57F7;
   // UNICODE_TO_GBK[6537] := 16#88CC;
   // UNICODE_TO_GBK[6538] := 16#57F8;
   // UNICODE_TO_GBK[6539] := 16#DBFC;
   // UNICODE_TO_GBK[6540] := 16#57F9;
   // UNICODE_TO_GBK[6541] := 16#C5E0;
   // UNICODE_TO_GBK[6542] := 16#57FA;
   // UNICODE_TO_GBK[6543] := 16#BBF9;
   // UNICODE_TO_GBK[6544] := 16#57FB;
   // UNICODE_TO_GBK[6545] := 16#88CD;
   // UNICODE_TO_GBK[6546] := 16#57FC;
   // UNICODE_TO_GBK[6547] := 16#88CE;
   // UNICODE_TO_GBK[6548] := 16#57FD;
   // UNICODE_TO_GBK[6549] := 16#DCA3;
   // UNICODE_TO_GBK[6550] := 16#57FE;
   // UNICODE_TO_GBK[6551] := 16#88CF;
   // UNICODE_TO_GBK[6552] := 16#57FF;
   // UNICODE_TO_GBK[6553] := 16#88D0;
   // UNICODE_TO_GBK[6554] := 16#5800;
   // UNICODE_TO_GBK[6555] := 16#DCA5;
   // UNICODE_TO_GBK[6556] := 16#5801;
   // UNICODE_TO_GBK[6557] := 16#88D1;
   // UNICODE_TO_GBK[6558] := 16#5802;
   // UNICODE_TO_GBK[6559] := 16#CCC3;
   // UNICODE_TO_GBK[6560] := 16#5803;
   // UNICODE_TO_GBK[6561] := 16#88D2;
   // UNICODE_TO_GBK[6562] := 16#5804;
   // UNICODE_TO_GBK[6563] := 16#88D3;
   // UNICODE_TO_GBK[6564] := 16#5805;
   // UNICODE_TO_GBK[6565] := 16#88D4;
   // UNICODE_TO_GBK[6566] := 16#5806;
   // UNICODE_TO_GBK[6567] := 16#B6D1;
   // UNICODE_TO_GBK[6568] := 16#5807;
   // UNICODE_TO_GBK[6569] := 16#DDC0;
   // UNICODE_TO_GBK[6570] := 16#5808;
   // UNICODE_TO_GBK[6571] := 16#88D5;
   // UNICODE_TO_GBK[6572] := 16#5809;
   // UNICODE_TO_GBK[6573] := 16#88D6;
   // UNICODE_TO_GBK[6574] := 16#580A;
   // UNICODE_TO_GBK[6575] := 16#88D7;
   // UNICODE_TO_GBK[6576] := 16#580B;
   // UNICODE_TO_GBK[6577] := 16#DCA1;
   // UNICODE_TO_GBK[6578] := 16#580C;
   // UNICODE_TO_GBK[6579] := 16#88D8;
   // UNICODE_TO_GBK[6580] := 16#580D;
   // UNICODE_TO_GBK[6581] := 16#DCA2;
   // UNICODE_TO_GBK[6582] := 16#580E;
   // UNICODE_TO_GBK[6583] := 16#88D9;
   // UNICODE_TO_GBK[6584] := 16#580F;
   // UNICODE_TO_GBK[6585] := 16#88DA;
   // UNICODE_TO_GBK[6586] := 16#5810;
   // UNICODE_TO_GBK[6587] := 16#88DB;
   // UNICODE_TO_GBK[6588] := 16#5811;
   // UNICODE_TO_GBK[6589] := 16#C7B5;
   // UNICODE_TO_GBK[6590] := 16#5812;
   // UNICODE_TO_GBK[6591] := 16#88DC;
   // UNICODE_TO_GBK[6592] := 16#5813;
   // UNICODE_TO_GBK[6593] := 16#88DD;
   // UNICODE_TO_GBK[6594] := 16#5814;
   // UNICODE_TO_GBK[6595] := 16#88DE;
   // UNICODE_TO_GBK[6596] := 16#5815;
   // UNICODE_TO_GBK[6597] := 16#B6E9;
   // UNICODE_TO_GBK[6598] := 16#5816;
   // UNICODE_TO_GBK[6599] := 16#88DF;
   // UNICODE_TO_GBK[6600] := 16#5817;
   // UNICODE_TO_GBK[6601] := 16#88E0;
   // UNICODE_TO_GBK[6602] := 16#5818;
   // UNICODE_TO_GBK[6603] := 16#88E1;
   // UNICODE_TO_GBK[6604] := 16#5819;
   // UNICODE_TO_GBK[6605] := 16#DCA7;
   // UNICODE_TO_GBK[6606] := 16#581A;
   // UNICODE_TO_GBK[6607] := 16#88E2;
   // UNICODE_TO_GBK[6608] := 16#581B;
   // UNICODE_TO_GBK[6609] := 16#88E3;
   // UNICODE_TO_GBK[6610] := 16#581C;
   // UNICODE_TO_GBK[6611] := 16#88E4;
   // UNICODE_TO_GBK[6612] := 16#581D;
   // UNICODE_TO_GBK[6613] := 16#88E5;
   // UNICODE_TO_GBK[6614] := 16#581E;
   // UNICODE_TO_GBK[6615] := 16#DCA6;
   // UNICODE_TO_GBK[6616] := 16#581F;
   // UNICODE_TO_GBK[6617] := 16#88E6;
   // UNICODE_TO_GBK[6618] := 16#5820;
   // UNICODE_TO_GBK[6619] := 16#DCA9;
   // UNICODE_TO_GBK[6620] := 16#5821;
   // UNICODE_TO_GBK[6621] := 16#B1A4;
   // UNICODE_TO_GBK[6622] := 16#5822;
   // UNICODE_TO_GBK[6623] := 16#88E7;
   // UNICODE_TO_GBK[6624] := 16#5823;
   // UNICODE_TO_GBK[6625] := 16#88E8;
   // UNICODE_TO_GBK[6626] := 16#5824;
   // UNICODE_TO_GBK[6627] := 16#B5CC;
   // UNICODE_TO_GBK[6628] := 16#5825;
   // UNICODE_TO_GBK[6629] := 16#88E9;
   // UNICODE_TO_GBK[6630] := 16#5826;
   // UNICODE_TO_GBK[6631] := 16#88EA;
   // UNICODE_TO_GBK[6632] := 16#5827;
   // UNICODE_TO_GBK[6633] := 16#88EB;
   // UNICODE_TO_GBK[6634] := 16#5828;
   // UNICODE_TO_GBK[6635] := 16#88EC;
   // UNICODE_TO_GBK[6636] := 16#5829;
   // UNICODE_TO_GBK[6637] := 16#88ED;
   // UNICODE_TO_GBK[6638] := 16#582A;
   // UNICODE_TO_GBK[6639] := 16#BFB0;
   // UNICODE_TO_GBK[6640] := 16#582B;
   // UNICODE_TO_GBK[6641] := 16#88EE;
   // UNICODE_TO_GBK[6642] := 16#582C;
   // UNICODE_TO_GBK[6643] := 16#88EF;
   // UNICODE_TO_GBK[6644] := 16#582D;
   // UNICODE_TO_GBK[6645] := 16#88F0;
   // UNICODE_TO_GBK[6646] := 16#582E;
   // UNICODE_TO_GBK[6647] := 16#88F1;
   // UNICODE_TO_GBK[6648] := 16#582F;
   // UNICODE_TO_GBK[6649] := 16#88F2;
   // UNICODE_TO_GBK[6650] := 16#5830;
   // UNICODE_TO_GBK[6651] := 16#D1DF;
   // UNICODE_TO_GBK[6652] := 16#5831;
   // UNICODE_TO_GBK[6653] := 16#88F3;
   // UNICODE_TO_GBK[6654] := 16#5832;
   // UNICODE_TO_GBK[6655] := 16#88F4;
   // UNICODE_TO_GBK[6656] := 16#5833;
   // UNICODE_TO_GBK[6657] := 16#88F5;
   // UNICODE_TO_GBK[6658] := 16#5834;
   // UNICODE_TO_GBK[6659] := 16#88F6;
   // UNICODE_TO_GBK[6660] := 16#5835;
   // UNICODE_TO_GBK[6661] := 16#B6C2;
   // UNICODE_TO_GBK[6662] := 16#5836;
   // UNICODE_TO_GBK[6663] := 16#88F7;
   // UNICODE_TO_GBK[6664] := 16#5837;
   // UNICODE_TO_GBK[6665] := 16#88F8;
   // UNICODE_TO_GBK[6666] := 16#5838;
   // UNICODE_TO_GBK[6667] := 16#88F9;
   // UNICODE_TO_GBK[6668] := 16#5839;
   // UNICODE_TO_GBK[6669] := 16#88FA;
   // UNICODE_TO_GBK[6670] := 16#583A;
   // UNICODE_TO_GBK[6671] := 16#88FB;
   // UNICODE_TO_GBK[6672] := 16#583B;
   // UNICODE_TO_GBK[6673] := 16#88FC;
   // UNICODE_TO_GBK[6674] := 16#583C;
   // UNICODE_TO_GBK[6675] := 16#88FD;
   // UNICODE_TO_GBK[6676] := 16#583D;
   // UNICODE_TO_GBK[6677] := 16#88FE;
   // UNICODE_TO_GBK[6678] := 16#583E;
   // UNICODE_TO_GBK[6679] := 16#8940;
   // UNICODE_TO_GBK[6680] := 16#583F;
   // UNICODE_TO_GBK[6681] := 16#8941;
   // UNICODE_TO_GBK[6682] := 16#5840;
   // UNICODE_TO_GBK[6683] := 16#8942;
   // UNICODE_TO_GBK[6684] := 16#5841;
   // UNICODE_TO_GBK[6685] := 16#8943;
   // UNICODE_TO_GBK[6686] := 16#5842;
   // UNICODE_TO_GBK[6687] := 16#8944;
   // UNICODE_TO_GBK[6688] := 16#5843;
   // UNICODE_TO_GBK[6689] := 16#8945;
   // UNICODE_TO_GBK[6690] := 16#5844;
   // UNICODE_TO_GBK[6691] := 16#DCA8;
   // UNICODE_TO_GBK[6692] := 16#5845;
   // UNICODE_TO_GBK[6693] := 16#8946;
   // UNICODE_TO_GBK[6694] := 16#5846;
   // UNICODE_TO_GBK[6695] := 16#8947;
   // UNICODE_TO_GBK[6696] := 16#5847;
   // UNICODE_TO_GBK[6697] := 16#8948;
   // UNICODE_TO_GBK[6698] := 16#5848;
   // UNICODE_TO_GBK[6699] := 16#8949;
   // UNICODE_TO_GBK[6700] := 16#5849;
   // UNICODE_TO_GBK[6701] := 16#894A;
   // UNICODE_TO_GBK[6702] := 16#584A;
   // UNICODE_TO_GBK[6703] := 16#894B;
   // UNICODE_TO_GBK[6704] := 16#584B;
   // UNICODE_TO_GBK[6705] := 16#894C;
   // UNICODE_TO_GBK[6706] := 16#584C;
   // UNICODE_TO_GBK[6707] := 16#CBFA;
   // UNICODE_TO_GBK[6708] := 16#584D;
   // UNICODE_TO_GBK[6709] := 16#EBF3;
   // UNICODE_TO_GBK[6710] := 16#584E;
   // UNICODE_TO_GBK[6711] := 16#894D;
   // UNICODE_TO_GBK[6712] := 16#584F;
   // UNICODE_TO_GBK[6713] := 16#894E;
   // UNICODE_TO_GBK[6714] := 16#5850;
   // UNICODE_TO_GBK[6715] := 16#894F;
   // UNICODE_TO_GBK[6716] := 16#5851;
   // UNICODE_TO_GBK[6717] := 16#CBDC;
   // UNICODE_TO_GBK[6718] := 16#5852;
   // UNICODE_TO_GBK[6719] := 16#8950;
   // UNICODE_TO_GBK[6720] := 16#5853;
   // UNICODE_TO_GBK[6721] := 16#8951;
   // UNICODE_TO_GBK[6722] := 16#5854;
   // UNICODE_TO_GBK[6723] := 16#CBFE;
   // UNICODE_TO_GBK[6724] := 16#5855;
   // UNICODE_TO_GBK[6725] := 16#8952;
   // UNICODE_TO_GBK[6726] := 16#5856;
   // UNICODE_TO_GBK[6727] := 16#8953;
   // UNICODE_TO_GBK[6728] := 16#5857;
   // UNICODE_TO_GBK[6729] := 16#8954;
   // UNICODE_TO_GBK[6730] := 16#5858;
   // UNICODE_TO_GBK[6731] := 16#CCC1;
   // UNICODE_TO_GBK[6732] := 16#5859;
   // UNICODE_TO_GBK[6733] := 16#8955;
   // UNICODE_TO_GBK[6734] := 16#585A;
   // UNICODE_TO_GBK[6735] := 16#8956;
   // UNICODE_TO_GBK[6736] := 16#585B;
   // UNICODE_TO_GBK[6737] := 16#8957;
   // UNICODE_TO_GBK[6738] := 16#585C;
   // UNICODE_TO_GBK[6739] := 16#8958;
   // UNICODE_TO_GBK[6740] := 16#585D;
   // UNICODE_TO_GBK[6741] := 16#8959;
   // UNICODE_TO_GBK[6742] := 16#585E;
   // UNICODE_TO_GBK[6743] := 16#C8FB;
   // UNICODE_TO_GBK[6744] := 16#585F;
   // UNICODE_TO_GBK[6745] := 16#895A;
   // UNICODE_TO_GBK[6746] := 16#5860;
   // UNICODE_TO_GBK[6747] := 16#895B;
   // UNICODE_TO_GBK[6748] := 16#5861;
   // UNICODE_TO_GBK[6749] := 16#895C;
   // UNICODE_TO_GBK[6750] := 16#5862;
   // UNICODE_TO_GBK[6751] := 16#895D;
   // UNICODE_TO_GBK[6752] := 16#5863;
   // UNICODE_TO_GBK[6753] := 16#895E;
   // UNICODE_TO_GBK[6754] := 16#5864;
   // UNICODE_TO_GBK[6755] := 16#895F;
   // UNICODE_TO_GBK[6756] := 16#5865;
   // UNICODE_TO_GBK[6757] := 16#DCAA;
   // UNICODE_TO_GBK[6758] := 16#5866;
   // UNICODE_TO_GBK[6759] := 16#8960;
   // UNICODE_TO_GBK[6760] := 16#5867;
   // UNICODE_TO_GBK[6761] := 16#8961;
   // UNICODE_TO_GBK[6762] := 16#5868;
   // UNICODE_TO_GBK[6763] := 16#8962;
   // UNICODE_TO_GBK[6764] := 16#5869;
   // UNICODE_TO_GBK[6765] := 16#8963;
   // UNICODE_TO_GBK[6766] := 16#586A;
   // UNICODE_TO_GBK[6767] := 16#8964;
   // UNICODE_TO_GBK[6768] := 16#586B;
   // UNICODE_TO_GBK[6769] := 16#CCEE;
   // UNICODE_TO_GBK[6770] := 16#586C;
   // UNICODE_TO_GBK[6771] := 16#DCAB;
   // UNICODE_TO_GBK[6772] := 16#586D;
   // UNICODE_TO_GBK[6773] := 16#8965;
   // UNICODE_TO_GBK[6774] := 16#586E;
   // UNICODE_TO_GBK[6775] := 16#8966;
   // UNICODE_TO_GBK[6776] := 16#586F;
   // UNICODE_TO_GBK[6777] := 16#8967;
   // UNICODE_TO_GBK[6778] := 16#5870;
   // UNICODE_TO_GBK[6779] := 16#8968;
   // UNICODE_TO_GBK[6780] := 16#5871;
   // UNICODE_TO_GBK[6781] := 16#8969;
   // UNICODE_TO_GBK[6782] := 16#5872;
   // UNICODE_TO_GBK[6783] := 16#896A;
   // UNICODE_TO_GBK[6784] := 16#5873;
   // UNICODE_TO_GBK[6785] := 16#896B;
   // UNICODE_TO_GBK[6786] := 16#5874;
   // UNICODE_TO_GBK[6787] := 16#896C;
   // UNICODE_TO_GBK[6788] := 16#5875;
   // UNICODE_TO_GBK[6789] := 16#896D;
   // UNICODE_TO_GBK[6790] := 16#5876;
   // UNICODE_TO_GBK[6791] := 16#896E;
   // UNICODE_TO_GBK[6792] := 16#5877;
   // UNICODE_TO_GBK[6793] := 16#896F;
   // UNICODE_TO_GBK[6794] := 16#5878;
   // UNICODE_TO_GBK[6795] := 16#8970;
   // UNICODE_TO_GBK[6796] := 16#5879;
   // UNICODE_TO_GBK[6797] := 16#8971;
   // UNICODE_TO_GBK[6798] := 16#587A;
   // UNICODE_TO_GBK[6799] := 16#8972;
   // UNICODE_TO_GBK[6800] := 16#587B;
   // UNICODE_TO_GBK[6801] := 16#8973;
   // UNICODE_TO_GBK[6802] := 16#587C;
   // UNICODE_TO_GBK[6803] := 16#8974;
   // UNICODE_TO_GBK[6804] := 16#587D;
   // UNICODE_TO_GBK[6805] := 16#8975;
   // UNICODE_TO_GBK[6806] := 16#587E;
   // UNICODE_TO_GBK[6807] := 16#DBD3;
   // UNICODE_TO_GBK[6808] := 16#587F;
   // UNICODE_TO_GBK[6809] := 16#8976;
   // UNICODE_TO_GBK[6810] := 16#5880;
   // UNICODE_TO_GBK[6811] := 16#DCAF;
   // UNICODE_TO_GBK[6812] := 16#5881;
   // UNICODE_TO_GBK[6813] := 16#DCAC;
   // UNICODE_TO_GBK[6814] := 16#5882;
   // UNICODE_TO_GBK[6815] := 16#8977;
   // UNICODE_TO_GBK[6816] := 16#5883;
   // UNICODE_TO_GBK[6817] := 16#BEB3;
   // UNICODE_TO_GBK[6818] := 16#5884;
   // UNICODE_TO_GBK[6819] := 16#8978;
   // UNICODE_TO_GBK[6820] := 16#5885;
   // UNICODE_TO_GBK[6821] := 16#CAFB;
   // UNICODE_TO_GBK[6822] := 16#5886;
   // UNICODE_TO_GBK[6823] := 16#8979;
   // UNICODE_TO_GBK[6824] := 16#5887;
   // UNICODE_TO_GBK[6825] := 16#897A;
   // UNICODE_TO_GBK[6826] := 16#5888;
   // UNICODE_TO_GBK[6827] := 16#897B;
   // UNICODE_TO_GBK[6828] := 16#5889;
   // UNICODE_TO_GBK[6829] := 16#DCAD;
   // UNICODE_TO_GBK[6830] := 16#588A;
   // UNICODE_TO_GBK[6831] := 16#897C;
   // UNICODE_TO_GBK[6832] := 16#588B;
   // UNICODE_TO_GBK[6833] := 16#897D;
   // UNICODE_TO_GBK[6834] := 16#588C;
   // UNICODE_TO_GBK[6835] := 16#897E;
   // UNICODE_TO_GBK[6836] := 16#588D;
   // UNICODE_TO_GBK[6837] := 16#8980;
   // UNICODE_TO_GBK[6838] := 16#588E;
   // UNICODE_TO_GBK[6839] := 16#8981;
   // UNICODE_TO_GBK[6840] := 16#588F;
   // UNICODE_TO_GBK[6841] := 16#8982;
   // UNICODE_TO_GBK[6842] := 16#5890;
   // UNICODE_TO_GBK[6843] := 16#8983;
   // UNICODE_TO_GBK[6844] := 16#5891;
   // UNICODE_TO_GBK[6845] := 16#8984;
   // UNICODE_TO_GBK[6846] := 16#5892;
   // UNICODE_TO_GBK[6847] := 16#C9CA;
   // UNICODE_TO_GBK[6848] := 16#5893;
   // UNICODE_TO_GBK[6849] := 16#C4B9;
   // UNICODE_TO_GBK[6850] := 16#5894;
   // UNICODE_TO_GBK[6851] := 16#8985;
   // UNICODE_TO_GBK[6852] := 16#5895;
   // UNICODE_TO_GBK[6853] := 16#8986;
   // UNICODE_TO_GBK[6854] := 16#5896;
   // UNICODE_TO_GBK[6855] := 16#8987;
   // UNICODE_TO_GBK[6856] := 16#5897;
   // UNICODE_TO_GBK[6857] := 16#8988;
   // UNICODE_TO_GBK[6858] := 16#5898;
   // UNICODE_TO_GBK[6859] := 16#8989;
   // UNICODE_TO_GBK[6860] := 16#5899;
   // UNICODE_TO_GBK[6861] := 16#C7BD;
   // UNICODE_TO_GBK[6862] := 16#589A;
   // UNICODE_TO_GBK[6863] := 16#DCAE;
   // UNICODE_TO_GBK[6864] := 16#589B;
   // UNICODE_TO_GBK[6865] := 16#898A;
   // UNICODE_TO_GBK[6866] := 16#589C;
   // UNICODE_TO_GBK[6867] := 16#898B;
   // UNICODE_TO_GBK[6868] := 16#589D;
   // UNICODE_TO_GBK[6869] := 16#898C;
   // UNICODE_TO_GBK[6870] := 16#589E;
   // UNICODE_TO_GBK[6871] := 16#D4F6;
   // UNICODE_TO_GBK[6872] := 16#589F;
   // UNICODE_TO_GBK[6873] := 16#D0E6;
   // UNICODE_TO_GBK[6874] := 16#58A0;
   // UNICODE_TO_GBK[6875] := 16#898D;
   // UNICODE_TO_GBK[6876] := 16#58A1;
   // UNICODE_TO_GBK[6877] := 16#898E;
   // UNICODE_TO_GBK[6878] := 16#58A2;
   // UNICODE_TO_GBK[6879] := 16#898F;
   // UNICODE_TO_GBK[6880] := 16#58A3;
   // UNICODE_TO_GBK[6881] := 16#8990;
   // UNICODE_TO_GBK[6882] := 16#58A4;
   // UNICODE_TO_GBK[6883] := 16#8991;
   // UNICODE_TO_GBK[6884] := 16#58A5;
   // UNICODE_TO_GBK[6885] := 16#8992;
   // UNICODE_TO_GBK[6886] := 16#58A6;
   // UNICODE_TO_GBK[6887] := 16#8993;
   // UNICODE_TO_GBK[6888] := 16#58A7;
   // UNICODE_TO_GBK[6889] := 16#8994;
   // UNICODE_TO_GBK[6890] := 16#58A8;
   // UNICODE_TO_GBK[6891] := 16#C4AB;
   // UNICODE_TO_GBK[6892] := 16#58A9;
   // UNICODE_TO_GBK[6893] := 16#B6D5;
   // UNICODE_TO_GBK[6894] := 16#58AA;
   // UNICODE_TO_GBK[6895] := 16#8995;
   // UNICODE_TO_GBK[6896] := 16#58AB;
   // UNICODE_TO_GBK[6897] := 16#8996;
   // UNICODE_TO_GBK[6898] := 16#58AC;
   // UNICODE_TO_GBK[6899] := 16#8997;
   // UNICODE_TO_GBK[6900] := 16#58AD;
   // UNICODE_TO_GBK[6901] := 16#8998;
   // UNICODE_TO_GBK[6902] := 16#58AE;
   // UNICODE_TO_GBK[6903] := 16#8999;
   // UNICODE_TO_GBK[6904] := 16#58AF;
   // UNICODE_TO_GBK[6905] := 16#899A;
   // UNICODE_TO_GBK[6906] := 16#58B0;
   // UNICODE_TO_GBK[6907] := 16#899B;
   // UNICODE_TO_GBK[6908] := 16#58B1;
   // UNICODE_TO_GBK[6909] := 16#899C;
   // UNICODE_TO_GBK[6910] := 16#58B2;
   // UNICODE_TO_GBK[6911] := 16#899D;
   // UNICODE_TO_GBK[6912] := 16#58B3;
   // UNICODE_TO_GBK[6913] := 16#899E;
   // UNICODE_TO_GBK[6914] := 16#58B4;
   // UNICODE_TO_GBK[6915] := 16#899F;
   // UNICODE_TO_GBK[6916] := 16#58B5;
   // UNICODE_TO_GBK[6917] := 16#89A0;
   // UNICODE_TO_GBK[6918] := 16#58B6;
   // UNICODE_TO_GBK[6919] := 16#89A1;
   // UNICODE_TO_GBK[6920] := 16#58B7;
   // UNICODE_TO_GBK[6921] := 16#89A2;
   // UNICODE_TO_GBK[6922] := 16#58B8;
   // UNICODE_TO_GBK[6923] := 16#89A3;
   // UNICODE_TO_GBK[6924] := 16#58B9;
   // UNICODE_TO_GBK[6925] := 16#89A4;
   // UNICODE_TO_GBK[6926] := 16#58BA;
   // UNICODE_TO_GBK[6927] := 16#89A5;
   // UNICODE_TO_GBK[6928] := 16#58BB;
   // UNICODE_TO_GBK[6929] := 16#89A6;
   // UNICODE_TO_GBK[6930] := 16#58BC;
   // UNICODE_TO_GBK[6931] := 16#DBD4;
   // UNICODE_TO_GBK[6932] := 16#58BD;
   // UNICODE_TO_GBK[6933] := 16#89A7;
   // UNICODE_TO_GBK[6934] := 16#58BE;
   // UNICODE_TO_GBK[6935] := 16#89A8;
   // UNICODE_TO_GBK[6936] := 16#58BF;
   // UNICODE_TO_GBK[6937] := 16#89A9;
   // UNICODE_TO_GBK[6938] := 16#58C0;
   // UNICODE_TO_GBK[6939] := 16#89AA;
   // UNICODE_TO_GBK[6940] := 16#58C1;
   // UNICODE_TO_GBK[6941] := 16#B1DA;
   // UNICODE_TO_GBK[6942] := 16#58C2;
   // UNICODE_TO_GBK[6943] := 16#89AB;
   // UNICODE_TO_GBK[6944] := 16#58C3;
   // UNICODE_TO_GBK[6945] := 16#89AC;
   // UNICODE_TO_GBK[6946] := 16#58C4;
   // UNICODE_TO_GBK[6947] := 16#89AD;
   // UNICODE_TO_GBK[6948] := 16#58C5;
   // UNICODE_TO_GBK[6949] := 16#DBD5;
   // UNICODE_TO_GBK[6950] := 16#58C6;
   // UNICODE_TO_GBK[6951] := 16#89AE;
   // UNICODE_TO_GBK[6952] := 16#58C7;
   // UNICODE_TO_GBK[6953] := 16#89AF;
   // UNICODE_TO_GBK[6954] := 16#58C8;
   // UNICODE_TO_GBK[6955] := 16#89B0;
   // UNICODE_TO_GBK[6956] := 16#58C9;
   // UNICODE_TO_GBK[6957] := 16#89B1;
   // UNICODE_TO_GBK[6958] := 16#58CA;
   // UNICODE_TO_GBK[6959] := 16#89B2;
   // UNICODE_TO_GBK[6960] := 16#58CB;
   // UNICODE_TO_GBK[6961] := 16#89B3;
   // UNICODE_TO_GBK[6962] := 16#58CC;
   // UNICODE_TO_GBK[6963] := 16#89B4;
   // UNICODE_TO_GBK[6964] := 16#58CD;
   // UNICODE_TO_GBK[6965] := 16#89B5;
   // UNICODE_TO_GBK[6966] := 16#58CE;
   // UNICODE_TO_GBK[6967] := 16#89B6;
   // UNICODE_TO_GBK[6968] := 16#58CF;
   // UNICODE_TO_GBK[6969] := 16#89B7;
   // UNICODE_TO_GBK[6970] := 16#58D0;
   // UNICODE_TO_GBK[6971] := 16#89B8;
   // UNICODE_TO_GBK[6972] := 16#58D1;
   // UNICODE_TO_GBK[6973] := 16#DBD6;
   // UNICODE_TO_GBK[6974] := 16#58D2;
   // UNICODE_TO_GBK[6975] := 16#89B9;
   // UNICODE_TO_GBK[6976] := 16#58D3;
   // UNICODE_TO_GBK[6977] := 16#89BA;
   // UNICODE_TO_GBK[6978] := 16#58D4;
   // UNICODE_TO_GBK[6979] := 16#89BB;
   // UNICODE_TO_GBK[6980] := 16#58D5;
   // UNICODE_TO_GBK[6981] := 16#BABE;
   // UNICODE_TO_GBK[6982] := 16#58D6;
   // UNICODE_TO_GBK[6983] := 16#89BC;
   // UNICODE_TO_GBK[6984] := 16#58D7;
   // UNICODE_TO_GBK[6985] := 16#89BD;
   // UNICODE_TO_GBK[6986] := 16#58D8;
   // UNICODE_TO_GBK[6987] := 16#89BE;
   // UNICODE_TO_GBK[6988] := 16#58D9;
   // UNICODE_TO_GBK[6989] := 16#89BF;
   // UNICODE_TO_GBK[6990] := 16#58DA;
   // UNICODE_TO_GBK[6991] := 16#89C0;
   // UNICODE_TO_GBK[6992] := 16#58DB;
   // UNICODE_TO_GBK[6993] := 16#89C1;
   // UNICODE_TO_GBK[6994] := 16#58DC;
   // UNICODE_TO_GBK[6995] := 16#89C2;
   // UNICODE_TO_GBK[6996] := 16#58DD;
   // UNICODE_TO_GBK[6997] := 16#89C3;
   // UNICODE_TO_GBK[6998] := 16#58DE;
   // UNICODE_TO_GBK[6999] := 16#89C4;
   // UNICODE_TO_GBK[7000] := 16#58DF;
   // UNICODE_TO_GBK[7001] := 16#89C5;
   // UNICODE_TO_GBK[7002] := 16#58E0;
   // UNICODE_TO_GBK[7003] := 16#89C6;
   // UNICODE_TO_GBK[7004] := 16#58E1;
   // UNICODE_TO_GBK[7005] := 16#89C7;
   // UNICODE_TO_GBK[7006] := 16#58E2;
   // UNICODE_TO_GBK[7007] := 16#89C8;
   // UNICODE_TO_GBK[7008] := 16#58E3;
   // UNICODE_TO_GBK[7009] := 16#89C9;
   // UNICODE_TO_GBK[7010] := 16#58E4;
   // UNICODE_TO_GBK[7011] := 16#C8C0;
   // UNICODE_TO_GBK[7012] := 16#58E5;
   // UNICODE_TO_GBK[7013] := 16#89CA;
   // UNICODE_TO_GBK[7014] := 16#58E6;
   // UNICODE_TO_GBK[7015] := 16#89CB;
   // UNICODE_TO_GBK[7016] := 16#58E7;
   // UNICODE_TO_GBK[7017] := 16#89CC;
   // UNICODE_TO_GBK[7018] := 16#58E8;
   // UNICODE_TO_GBK[7019] := 16#89CD;
   // UNICODE_TO_GBK[7020] := 16#58E9;
   // UNICODE_TO_GBK[7021] := 16#89CE;
   // UNICODE_TO_GBK[7022] := 16#58EA;
   // UNICODE_TO_GBK[7023] := 16#89CF;
   // UNICODE_TO_GBK[7024] := 16#58EB;
   // UNICODE_TO_GBK[7025] := 16#CABF;
   // UNICODE_TO_GBK[7026] := 16#58EC;
   // UNICODE_TO_GBK[7027] := 16#C8C9;
   // UNICODE_TO_GBK[7028] := 16#58ED;
   // UNICODE_TO_GBK[7029] := 16#89D0;
   // UNICODE_TO_GBK[7030] := 16#58EE;
   // UNICODE_TO_GBK[7031] := 16#D7B3;
   // UNICODE_TO_GBK[7032] := 16#58EF;
   // UNICODE_TO_GBK[7033] := 16#89D1;
   // UNICODE_TO_GBK[7034] := 16#58F0;
   // UNICODE_TO_GBK[7035] := 16#C9F9;
   // UNICODE_TO_GBK[7036] := 16#58F1;
   // UNICODE_TO_GBK[7037] := 16#89D2;
   // UNICODE_TO_GBK[7038] := 16#58F2;
   // UNICODE_TO_GBK[7039] := 16#89D3;
   // UNICODE_TO_GBK[7040] := 16#58F3;
   // UNICODE_TO_GBK[7041] := 16#BFC7;
   // UNICODE_TO_GBK[7042] := 16#58F4;
   // UNICODE_TO_GBK[7043] := 16#89D4;
   // UNICODE_TO_GBK[7044] := 16#58F5;
   // UNICODE_TO_GBK[7045] := 16#89D5;
   // UNICODE_TO_GBK[7046] := 16#58F6;
   // UNICODE_TO_GBK[7047] := 16#BAF8;
   // UNICODE_TO_GBK[7048] := 16#58F7;
   // UNICODE_TO_GBK[7049] := 16#89D6;
   // UNICODE_TO_GBK[7050] := 16#58F8;
   // UNICODE_TO_GBK[7051] := 16#89D7;
   // UNICODE_TO_GBK[7052] := 16#58F9;
   // UNICODE_TO_GBK[7053] := 16#D2BC;
   // UNICODE_TO_GBK[7054] := 16#58FA;
   // UNICODE_TO_GBK[7055] := 16#89D8;
   // UNICODE_TO_GBK[7056] := 16#58FB;
   // UNICODE_TO_GBK[7057] := 16#89D9;
   // UNICODE_TO_GBK[7058] := 16#58FC;
   // UNICODE_TO_GBK[7059] := 16#89DA;
   // UNICODE_TO_GBK[7060] := 16#58FD;
   // UNICODE_TO_GBK[7061] := 16#89DB;
   // UNICODE_TO_GBK[7062] := 16#58FE;
   // UNICODE_TO_GBK[7063] := 16#89DC;
   // UNICODE_TO_GBK[7064] := 16#58FF;
   // UNICODE_TO_GBK[7065] := 16#89DD;
   // UNICODE_TO_GBK[7066] := 16#5900;
   // UNICODE_TO_GBK[7067] := 16#89DE;
   // UNICODE_TO_GBK[7068] := 16#5901;
   // UNICODE_TO_GBK[7069] := 16#89DF;
   // UNICODE_TO_GBK[7070] := 16#5902;
   // UNICODE_TO_GBK[7071] := 16#E2BA;
   // UNICODE_TO_GBK[7072] := 16#5903;
   // UNICODE_TO_GBK[7073] := 16#89E0;
   // UNICODE_TO_GBK[7074] := 16#5904;
   // UNICODE_TO_GBK[7075] := 16#B4A6;
   // UNICODE_TO_GBK[7076] := 16#5905;
   // UNICODE_TO_GBK[7077] := 16#89E1;
   // UNICODE_TO_GBK[7078] := 16#5906;
   // UNICODE_TO_GBK[7079] := 16#89E2;
   // UNICODE_TO_GBK[7080] := 16#5907;
   // UNICODE_TO_GBK[7081] := 16#B1B8;
   // UNICODE_TO_GBK[7082] := 16#5908;
   // UNICODE_TO_GBK[7083] := 16#89E3;
   // UNICODE_TO_GBK[7084] := 16#5909;
   // UNICODE_TO_GBK[7085] := 16#89E4;
   // UNICODE_TO_GBK[7086] := 16#590A;
   // UNICODE_TO_GBK[7087] := 16#89E5;
   // UNICODE_TO_GBK[7088] := 16#590B;
   // UNICODE_TO_GBK[7089] := 16#89E6;
   // UNICODE_TO_GBK[7090] := 16#590C;
   // UNICODE_TO_GBK[7091] := 16#89E7;
   // UNICODE_TO_GBK[7092] := 16#590D;
   // UNICODE_TO_GBK[7093] := 16#B8B4;
   // UNICODE_TO_GBK[7094] := 16#590E;
   // UNICODE_TO_GBK[7095] := 16#89E8;
   // UNICODE_TO_GBK[7096] := 16#590F;
   // UNICODE_TO_GBK[7097] := 16#CFC4;
   // UNICODE_TO_GBK[7098] := 16#5910;
   // UNICODE_TO_GBK[7099] := 16#89E9;
   // UNICODE_TO_GBK[7100] := 16#5911;
   // UNICODE_TO_GBK[7101] := 16#89EA;
   // UNICODE_TO_GBK[7102] := 16#5912;
   // UNICODE_TO_GBK[7103] := 16#89EB;
   // UNICODE_TO_GBK[7104] := 16#5913;
   // UNICODE_TO_GBK[7105] := 16#89EC;
   // UNICODE_TO_GBK[7106] := 16#5914;
   // UNICODE_TO_GBK[7107] := 16#D9E7;
   // UNICODE_TO_GBK[7108] := 16#5915;
   // UNICODE_TO_GBK[7109] := 16#CFA6;
   // UNICODE_TO_GBK[7110] := 16#5916;
   // UNICODE_TO_GBK[7111] := 16#CDE2;
   // UNICODE_TO_GBK[7112] := 16#5917;
   // UNICODE_TO_GBK[7113] := 16#89ED;
   // UNICODE_TO_GBK[7114] := 16#5918;
   // UNICODE_TO_GBK[7115] := 16#89EE;
   // UNICODE_TO_GBK[7116] := 16#5919;
   // UNICODE_TO_GBK[7117] := 16#D9ED;
   // UNICODE_TO_GBK[7118] := 16#591A;
   // UNICODE_TO_GBK[7119] := 16#B6E0;
   // UNICODE_TO_GBK[7120] := 16#591B;
   // UNICODE_TO_GBK[7121] := 16#89EF;
   // UNICODE_TO_GBK[7122] := 16#591C;
   // UNICODE_TO_GBK[7123] := 16#D2B9;
   // UNICODE_TO_GBK[7124] := 16#591D;
   // UNICODE_TO_GBK[7125] := 16#89F0;
   // UNICODE_TO_GBK[7126] := 16#591E;
   // UNICODE_TO_GBK[7127] := 16#89F1;
   // UNICODE_TO_GBK[7128] := 16#591F;
   // UNICODE_TO_GBK[7129] := 16#B9BB;
   // UNICODE_TO_GBK[7130] := 16#5920;
   // UNICODE_TO_GBK[7131] := 16#89F2;
   // UNICODE_TO_GBK[7132] := 16#5921;
   // UNICODE_TO_GBK[7133] := 16#89F3;
   // UNICODE_TO_GBK[7134] := 16#5922;
   // UNICODE_TO_GBK[7135] := 16#89F4;
   // UNICODE_TO_GBK[7136] := 16#5923;
   // UNICODE_TO_GBK[7137] := 16#89F5;
   // UNICODE_TO_GBK[7138] := 16#5924;
   // UNICODE_TO_GBK[7139] := 16#E2B9;
   // UNICODE_TO_GBK[7140] := 16#5925;
   // UNICODE_TO_GBK[7141] := 16#E2B7;
   // UNICODE_TO_GBK[7142] := 16#5926;
   // UNICODE_TO_GBK[7143] := 16#89F6;
   // UNICODE_TO_GBK[7144] := 16#5927;
   // UNICODE_TO_GBK[7145] := 16#B4F3;
   // UNICODE_TO_GBK[7146] := 16#5928;
   // UNICODE_TO_GBK[7147] := 16#89F7;
   // UNICODE_TO_GBK[7148] := 16#5929;
   // UNICODE_TO_GBK[7149] := 16#CCEC;
   // UNICODE_TO_GBK[7150] := 16#592A;
   // UNICODE_TO_GBK[7151] := 16#CCAB;
   // UNICODE_TO_GBK[7152] := 16#592B;
   // UNICODE_TO_GBK[7153] := 16#B7F2;
   // UNICODE_TO_GBK[7154] := 16#592C;
   // UNICODE_TO_GBK[7155] := 16#89F8;
   // UNICODE_TO_GBK[7156] := 16#592D;
   // UNICODE_TO_GBK[7157] := 16#D8B2;
   // UNICODE_TO_GBK[7158] := 16#592E;
   // UNICODE_TO_GBK[7159] := 16#D1EB;
   // UNICODE_TO_GBK[7160] := 16#592F;
   // UNICODE_TO_GBK[7161] := 16#BABB;
   // UNICODE_TO_GBK[7162] := 16#5930;
   // UNICODE_TO_GBK[7163] := 16#89F9;
   // UNICODE_TO_GBK[7164] := 16#5931;
   // UNICODE_TO_GBK[7165] := 16#CAA7;
   // UNICODE_TO_GBK[7166] := 16#5932;
   // UNICODE_TO_GBK[7167] := 16#89FA;
   // UNICODE_TO_GBK[7168] := 16#5933;
   // UNICODE_TO_GBK[7169] := 16#89FB;
   // UNICODE_TO_GBK[7170] := 16#5934;
   // UNICODE_TO_GBK[7171] := 16#CDB7;
   // UNICODE_TO_GBK[7172] := 16#5935;
   // UNICODE_TO_GBK[7173] := 16#89FC;
   // UNICODE_TO_GBK[7174] := 16#5936;
   // UNICODE_TO_GBK[7175] := 16#89FD;
   // UNICODE_TO_GBK[7176] := 16#5937;
   // UNICODE_TO_GBK[7177] := 16#D2C4;
   // UNICODE_TO_GBK[7178] := 16#5938;
   // UNICODE_TO_GBK[7179] := 16#BFE4;
   // UNICODE_TO_GBK[7180] := 16#5939;
   // UNICODE_TO_GBK[7181] := 16#BCD0;
   // UNICODE_TO_GBK[7182] := 16#593A;
   // UNICODE_TO_GBK[7183] := 16#B6E1;
   // UNICODE_TO_GBK[7184] := 16#593B;
   // UNICODE_TO_GBK[7185] := 16#89FE;
   // UNICODE_TO_GBK[7186] := 16#593C;
   // UNICODE_TO_GBK[7187] := 16#DEC5;
   // UNICODE_TO_GBK[7188] := 16#593D;
   // UNICODE_TO_GBK[7189] := 16#8A40;
   // UNICODE_TO_GBK[7190] := 16#593E;
   // UNICODE_TO_GBK[7191] := 16#8A41;
   // UNICODE_TO_GBK[7192] := 16#593F;
   // UNICODE_TO_GBK[7193] := 16#8A42;
   // UNICODE_TO_GBK[7194] := 16#5940;
   // UNICODE_TO_GBK[7195] := 16#8A43;
   // UNICODE_TO_GBK[7196] := 16#5941;
   // UNICODE_TO_GBK[7197] := 16#DEC6;
   // UNICODE_TO_GBK[7198] := 16#5942;
   // UNICODE_TO_GBK[7199] := 16#DBBC;
   // UNICODE_TO_GBK[7200] := 16#5943;
   // UNICODE_TO_GBK[7201] := 16#8A44;
   // UNICODE_TO_GBK[7202] := 16#5944;
   // UNICODE_TO_GBK[7203] := 16#D1D9;
   // UNICODE_TO_GBK[7204] := 16#5945;
   // UNICODE_TO_GBK[7205] := 16#8A45;
   // UNICODE_TO_GBK[7206] := 16#5946;
   // UNICODE_TO_GBK[7207] := 16#8A46;
   // UNICODE_TO_GBK[7208] := 16#5947;
   // UNICODE_TO_GBK[7209] := 16#C6E6;
   // UNICODE_TO_GBK[7210] := 16#5948;
   // UNICODE_TO_GBK[7211] := 16#C4CE;
   // UNICODE_TO_GBK[7212] := 16#5949;
   // UNICODE_TO_GBK[7213] := 16#B7EE;
   // UNICODE_TO_GBK[7214] := 16#594A;
   // UNICODE_TO_GBK[7215] := 16#8A47;
   // UNICODE_TO_GBK[7216] := 16#594B;
   // UNICODE_TO_GBK[7217] := 16#B7DC;
   // UNICODE_TO_GBK[7218] := 16#594C;
   // UNICODE_TO_GBK[7219] := 16#8A48;
   // UNICODE_TO_GBK[7220] := 16#594D;
   // UNICODE_TO_GBK[7221] := 16#8A49;
   // UNICODE_TO_GBK[7222] := 16#594E;
   // UNICODE_TO_GBK[7223] := 16#BFFC;
   // UNICODE_TO_GBK[7224] := 16#594F;
   // UNICODE_TO_GBK[7225] := 16#D7E0;
   // UNICODE_TO_GBK[7226] := 16#5950;
   // UNICODE_TO_GBK[7227] := 16#8A4A;
   // UNICODE_TO_GBK[7228] := 16#5951;
   // UNICODE_TO_GBK[7229] := 16#C6F5;
   // UNICODE_TO_GBK[7230] := 16#5952;
   // UNICODE_TO_GBK[7231] := 16#8A4B;
   // UNICODE_TO_GBK[7232] := 16#5953;
   // UNICODE_TO_GBK[7233] := 16#8A4C;
   // UNICODE_TO_GBK[7234] := 16#5954;
   // UNICODE_TO_GBK[7235] := 16#B1BC;
   // UNICODE_TO_GBK[7236] := 16#5955;
   // UNICODE_TO_GBK[7237] := 16#DEC8;
   // UNICODE_TO_GBK[7238] := 16#5956;
   // UNICODE_TO_GBK[7239] := 16#BDB1;
   // UNICODE_TO_GBK[7240] := 16#5957;
   // UNICODE_TO_GBK[7241] := 16#CCD7;
   // UNICODE_TO_GBK[7242] := 16#5958;
   // UNICODE_TO_GBK[7243] := 16#DECA;
   // UNICODE_TO_GBK[7244] := 16#5959;
   // UNICODE_TO_GBK[7245] := 16#8A4D;
   // UNICODE_TO_GBK[7246] := 16#595A;
   // UNICODE_TO_GBK[7247] := 16#DEC9;
   // UNICODE_TO_GBK[7248] := 16#595B;
   // UNICODE_TO_GBK[7249] := 16#8A4E;
   // UNICODE_TO_GBK[7250] := 16#595C;
   // UNICODE_TO_GBK[7251] := 16#8A4F;
   // UNICODE_TO_GBK[7252] := 16#595D;
   // UNICODE_TO_GBK[7253] := 16#8A50;
   // UNICODE_TO_GBK[7254] := 16#595E;
   // UNICODE_TO_GBK[7255] := 16#8A51;
   // UNICODE_TO_GBK[7256] := 16#595F;
   // UNICODE_TO_GBK[7257] := 16#8A52;
